   1:  PR[GP1:91,1] = PR[GP1:90,1] + 82.412;
   1:  PR[GP1:91,2] = PR[GP1:90,2] + 125.667;
   1:L PR[91] 10mm/sec FINE;
   1:  PR[GP1:91,1] = PR[GP1:90,1] + 79.591;
   1:  PR[GP1:91,2] = PR[GP1:90,2] + 126.103;
   1:L PR[91] 10mm/sec FINE;
   1:  PR[GP1:91,1] = PR[GP1:90,1] + 77.896;
   1:  PR[GP1:91,2] = PR[GP1:90,2] + 126.057;
   1:L PR[91] 10mm/sec FINE;
   1:  PR[GP1:91,1] = PR[GP1:90,1] + 75.790;
   1:  PR[GP1:91,2] = PR[GP1:90,2] + 125.965;
   1:L PR[91] 10mm/sec FINE;
   1:  PR[GP1:91,1] = PR[GP1:90,1] + 72.240;
   1:  PR[GP1:91,2] = PR[GP1:90,2] + 125.093;
   1:L PR[91] 10mm/sec FINE;
   1:  PR[GP1:91,1] = PR[GP1:90,1] + 68.979;
   1:  PR[GP1:91,2] = PR[GP1:90,2] + 123.554;
   1:L PR[91] 10mm/sec FINE;
   1:  PR[GP1:91,1] = PR[GP1:90,1] + 67.464;
   1:  PR[GP1:91,2] = PR[GP1:90,2] + 122.423;
   1:L PR[91] 10mm/sec FINE;
   1:  PR[GP1:91,1] = PR[GP1:90,1] + 66.133;
   1:  PR[GP1:91,2] = PR[GP1:90,2] + 121.415;
   1:L PR[91] 10mm/sec FINE;
   1:  PR[GP1:91,1] = PR[GP1:90,1] + 63.816;
   1:  PR[GP1:91,2] = PR[GP1:90,2] + 118.763;
   1:L PR[91] 10mm/sec FINE;
   1:  PR[GP1:91,1] = PR[GP1:90,1] + 62.107;
   1:  PR[GP1:91,2] = PR[GP1:90,2] + 115.709;
   1:L PR[91] 10mm/sec FINE;
   1:  PR[GP1:91,1] = PR[GP1:90,1] + 61.054;
   1:  PR[GP1:91,2] = PR[GP1:90,2] + 112.384;
   1:L PR[91] 10mm/sec FINE;
   1:  PR[GP1:91,1] = PR[GP1:90,1] + 60.750;
   1:  PR[GP1:91,2] = PR[GP1:90,2] + 108.893;
   1:L PR[91] 10mm/sec FINE;
   1:  PR[GP1:91,1] = PR[GP1:90,1] + 60.970;
   1:  PR[GP1:91,2] = PR[GP1:90,2] + 107.084;
   1:L PR[91] 10mm/sec FINE;
   1:  PR[GP1:91,1] = PR[GP1:90,1] + 61.204;
   1:  PR[GP1:91,2] = PR[GP1:90,2] + 105.365;
   1:L PR[91] 10mm/sec FINE;
   1:  PR[GP1:91,1] = PR[GP1:90,1] + 62.339;
   1:  PR[GP1:91,2] = PR[GP1:90,2] + 101.980;
   1:L PR[91] 10mm/sec FINE;
   1:  PR[GP1:91,1] = PR[GP1:90,1] + 63.029;
   1:  PR[GP1:91,2] = PR[GP1:90,2] + 100.795;
   1:L PR[91] 10mm/sec FINE;
   1:  PR[GP1:91,1] = PR[GP1:90,1] + 64.194;
   1:  PR[GP1:91,2] = PR[GP1:90,2] + 98.846;
   1:L PR[91] 10mm/sec FINE;
   1:  PR[GP1:91,1] = PR[GP1:90,1] + 64.821;
   1:  PR[GP1:91,2] = PR[GP1:90,2] + 98.140;
   1:L PR[91] 10mm/sec FINE;
   1:  PR[GP1:91,1] = PR[GP1:90,1] + 66.690;
   1:  PR[GP1:91,2] = PR[GP1:90,2] + 96.102;
   1:L PR[91] 10mm/sec FINE;
   1:  PR[GP1:91,1] = PR[GP1:90,1] + 68.560;
   1:  PR[GP1:91,2] = PR[GP1:90,2] + 94.729;
   1:L PR[91] 10mm/sec FINE;
   1:  PR[GP1:91,1] = PR[GP1:90,1] + 69.814;
   1:  PR[GP1:91,2] = PR[GP1:90,2] + 93.845;
   1:L PR[91] 10mm/sec FINE;
   1:  PR[GP1:91,1] = PR[GP1:90,1] + 70.348;
   1:  PR[GP1:91,2] = PR[GP1:90,2] + 93.651;
   1:  PR[GP1:91,3] = PR[GP1:90,3] + 22.900;
   1:L PR[91] 10mm/sec FINE;
   1:  PR[GP1:91,1] = PR[GP1:90,1] + 72.452;
   1:  PR[GP1:91,2] = PR[GP1:90,2] + 92.683;
   1:L PR[91] 10mm/sec FINE;
   1:  PR[GP1:91,1] = PR[GP1:90,1] + 74.148;
   1:  PR[GP1:91,2] = PR[GP1:90,2] + 91.983;
   1:L PR[91] 10mm/sec FINE;
   1:  PR[GP1:91,1] = PR[GP1:90,1] + 75.437;
   1:  PR[GP1:91,2] = PR[GP1:90,2] + 91.661;
   1:L PR[91] 10mm/sec FINE;
   1:  PR[GP1:91,1] = PR[GP1:90,1] + 78.330;
   1:  PR[GP1:91,2] = PR[GP1:90,2] + 91.079;
   1:L PR[91] 10mm/sec FINE;
   1:  PR[GP1:91,1] = PR[GP1:90,1] + 82.087;
   1:  PR[GP1:91,2] = PR[GP1:90,2] + 90.960;
   1:L PR[91] 10mm/sec FINE;
   1:  PR[GP1:91,1] = PR[GP1:90,1] + 83.731;
   1:  PR[GP1:91,2] = PR[GP1:90,2] + 91.115;
   1:L PR[91] 10mm/sec FINE;
   1:  PR[GP1:91,1] = PR[GP1:90,1] + 85.492;
   1:  PR[GP1:91,2] = PR[GP1:90,2] + 91.389;
   1:L PR[91] 10mm/sec FINE;
   1:  PR[GP1:91,1] = PR[GP1:90,1] + 88.274;
   1:  PR[GP1:91,2] = PR[GP1:90,2] + 92.183;
   1:L PR[91] 10mm/sec FINE;
   1:  PR[GP1:91,1] = PR[GP1:90,1] + 88.650;
   1:  PR[GP1:91,2] = PR[GP1:90,2] + 92.270;
   1:L PR[91] 10mm/sec FINE;
   1:  PR[GP1:91,1] = PR[GP1:90,1] + 88.838;
   1:  PR[GP1:91,2] = PR[GP1:90,2] + 92.342;
   1:L PR[91] 10mm/sec FINE;
   1:  PR[GP1:91,1] = PR[GP1:90,1] + 91.683;
   1:  PR[GP1:91,2] = PR[GP1:90,2] + 93.587;
   1:L PR[91] 10mm/sec FINE;
   1:  PR[GP1:91,1] = PR[GP1:90,1] + 93.071;
   1:  PR[GP1:91,2] = PR[GP1:90,2] + 94.392;
   1:L PR[91] 10mm/sec FINE;
   1:  PR[GP1:91,1] = PR[GP1:90,1] + 94.027;
   1:  PR[GP1:91,2] = PR[GP1:90,2] + 95.076;
   1:L PR[91] 10mm/sec FINE;
   1:  PR[GP1:91,1] = PR[GP1:90,1] + 94.243;
   1:  PR[GP1:91,2] = PR[GP1:90,2] + 95.199;
   1:L PR[91] 10mm/sec FINE;
   1:  PR[GP1:91,1] = PR[GP1:90,1] + 94.681;
   1:  PR[GP1:91,2] = PR[GP1:90,2] + 95.389;
   1:L PR[91] 10mm/sec FINE;
   1:  PR[GP1:91,1] = PR[GP1:90,1] + 95.163;
   1:  PR[GP1:91,2] = PR[GP1:90,2] + 95.421;
   1:L PR[91] 10mm/sec FINE;
   1:  PR[GP1:91,1] = PR[GP1:90,1] + 95.410;
   1:  PR[GP1:91,2] = PR[GP1:90,2] + 95.407;
   1:L PR[91] 10mm/sec FINE;
   1:  PR[GP1:91,1] = PR[GP1:90,1] + 95.904;
   1:  PR[GP1:91,2] = PR[GP1:90,2] + 95.271;
   1:L PR[91] 10mm/sec FINE;
   1:  PR[GP1:91,1] = PR[GP1:90,1] + 96.393;
   1:  PR[GP1:91,2] = PR[GP1:90,2] + 94.958;
   1:L PR[91] 10mm/sec FINE;
   1:  PR[GP1:91,1] = PR[GP1:90,1] + 97.232;
   1:  PR[GP1:91,2] = PR[GP1:90,2] + 94.289;
   1:L PR[91] 10mm/sec FINE;
   1:  PR[GP1:91,1] = PR[GP1:90,1] + 97.918;
   1:  PR[GP1:91,2] = PR[GP1:90,2] + 93.780;
   1:L PR[91] 10mm/sec FINE;
   1:  PR[GP1:91,1] = PR[GP1:90,1] + 98.083;
   1:  PR[GP1:91,2] = PR[GP1:90,2] + 93.673;
   1:L PR[91] 10mm/sec FINE;
   1:  PR[GP1:91,1] = PR[GP1:90,1] + 100.385;
   1:  PR[GP1:91,2] = PR[GP1:90,2] + 92.371;
   1:L PR[91] 10mm/sec FINE;
   1:  PR[GP1:91,1] = PR[GP1:90,1] + 102.853;
   1:  PR[GP1:91,2] = PR[GP1:90,2] + 91.430;
   1:L PR[91] 10mm/sec FINE;
   1:  PR[GP1:91,1] = PR[GP1:90,1] + 103.095;
   1:  PR[GP1:91,2] = PR[GP1:90,2] + 91.369;
   1:L PR[91] 10mm/sec FINE;
   1:  PR[GP1:91,1] = PR[GP1:90,1] + 105.479;
   1:  PR[GP1:91,2] = PR[GP1:90,2] + 90.840;
   1:L PR[91] 10mm/sec FINE;
   1:  PR[GP1:91,1] = PR[GP1:90,1] + 106.414;
   1:  PR[GP1:91,2] = PR[GP1:90,2] + 90.749;
   1:L PR[91] 10mm/sec FINE;
   1:  PR[GP1:91,1] = PR[GP1:90,1] + 108.189;
   1:  PR[GP1:91,2] = PR[GP1:90,2] + 90.619;
   1:L PR[91] 10mm/sec FINE;
   1:  PR[GP1:91,1] = PR[GP1:90,1] + 110.016;
   1:  PR[GP1:91,2] = PR[GP1:90,2] + 90.709;
   1:L PR[91] 10mm/sec FINE;
   1:  PR[GP1:91,1] = PR[GP1:90,1] + 110.931;
   1:  PR[GP1:91,2] = PR[GP1:90,2] + 90.772;
   1:L PR[91] 10mm/sec FINE;
   1:  PR[GP1:91,1] = PR[GP1:90,1] + 113.661;
   1:  PR[GP1:91,2] = PR[GP1:90,2] + 91.296;
   1:L PR[91] 10mm/sec FINE;
   1:  PR[GP1:91,1] = PR[GP1:90,1] + 116.348;
   1:  PR[GP1:91,2] = PR[GP1:90,2] + 92.156;
   1:L PR[91] 10mm/sec FINE;
   1:  PR[GP1:91,1] = PR[GP1:90,1] + 117.613;
   1:  PR[GP1:91,2] = PR[GP1:90,2] + 92.742;
   1:L PR[91] 10mm/sec FINE;
   1:  PR[GP1:91,1] = PR[GP1:90,1] + 118.911;
   1:  PR[GP1:91,2] = PR[GP1:90,2] + 93.369;
   1:L PR[91] 10mm/sec FINE;
   1:  PR[GP1:91,1] = PR[GP1:90,1] + 121.140;
   1:  PR[GP1:91,2] = PR[GP1:90,2] + 94.819;
   1:L PR[91] 10mm/sec FINE;
   1:  PR[GP1:91,1] = PR[GP1:90,1] + 121.299;
   1:  PR[GP1:91,2] = PR[GP1:90,2] + 94.926;
   1:L PR[91] 10mm/sec FINE;
   1:  PR[GP1:91,1] = PR[GP1:90,1] + 123.469;
   1:  PR[GP1:91,2] = PR[GP1:90,2] + 96.788;
   1:L PR[91] 10mm/sec FINE;
   1:  PR[GP1:91,1] = PR[GP1:90,1] + 125.338;
   1:  PR[GP1:91,2] = PR[GP1:90,2] + 98.930;
   1:L PR[91] 10mm/sec FINE;
   1:  PR[GP1:91,1] = PR[GP1:90,1] + 126.852;
   1:  PR[GP1:91,2] = PR[GP1:90,2] + 101.311;
   1:L PR[91] 10mm/sec FINE;
   1:  PR[GP1:91,1] = PR[GP1:90,1] + 127.765;
   1:  PR[GP1:91,2] = PR[GP1:90,2] + 103.396;
   1:L PR[91] 10mm/sec FINE;
   1:  PR[GP1:91,1] = PR[GP1:90,1] + 127.971;
   1:  PR[GP1:91,2] = PR[GP1:90,2] + 103.876;
   1:L PR[91] 10mm/sec FINE;
   1:  PR[GP1:91,1] = PR[GP1:90,1] + 128.656;
   1:  PR[GP1:91,2] = PR[GP1:90,2] + 106.564;
   1:L PR[91] 10mm/sec FINE;
   1:  PR[GP1:91,1] = PR[GP1:90,1] + 128.872;
   1:  PR[GP1:91,2] = PR[GP1:90,2] + 109.304;
   1:L PR[91] 10mm/sec FINE;
   1:  PR[GP1:91,1] = PR[GP1:90,1] + 128.474;
   1:  PR[GP1:91,2] = PR[GP1:90,2] + 112.731;
   1:L PR[91] 10mm/sec FINE;
   1:  PR[GP1:91,1] = PR[GP1:90,1] + 127.375;
   1:  PR[GP1:91,2] = PR[GP1:90,2] + 116.010;
   1:L PR[91] 10mm/sec FINE;
   1:  PR[GP1:91,1] = PR[GP1:90,1] + 125.589;
   1:  PR[GP1:91,2] = PR[GP1:90,2] + 119.007;
   1:L PR[91] 10mm/sec FINE;
   1:  PR[GP1:91,1] = PR[GP1:90,1] + 123.186;
   1:  PR[GP1:91,2] = PR[GP1:90,2] + 121.609;
   1:L PR[91] 10mm/sec FINE;
   1:  PR[GP1:91,1] = PR[GP1:90,1] + 120.265;
   1:  PR[GP1:91,2] = PR[GP1:90,2] + 123.714;
   1:L PR[91] 10mm/sec FINE;
   1:  PR[GP1:91,1] = PR[GP1:90,1] + 116.935;
   1:  PR[GP1:91,2] = PR[GP1:90,2] + 125.215;
   1:L PR[91] 10mm/sec FINE;
   1:  PR[GP1:91,1] = PR[GP1:90,1] + 113.317;
   1:  PR[GP1:91,2] = PR[GP1:90,2] + 126.080;
   1:L PR[91] 10mm/sec FINE;
   1:  PR[GP1:91,1] = PR[GP1:90,1] + 112.605;
   1:  PR[GP1:91,2] = PR[GP1:90,2] + 126.119;
   1:L PR[91] 10mm/sec FINE;
   1:  PR[GP1:91,1] = PR[GP1:90,1] + 109.577;
   1:  PR[GP1:91,2] = PR[GP1:90,2] + 126.268;
   1:L PR[91] 10mm/sec FINE;
   1:  PR[GP1:91,1] = PR[GP1:90,1] + 105.878;
   1:  PR[GP1:91,2] = PR[GP1:90,2] + 125.766;
   1:L PR[91] 10mm/sec FINE;
   1:  PR[GP1:91,1] = PR[GP1:90,1] + 102.315;
   1:  PR[GP1:91,2] = PR[GP1:90,2] + 124.617;
   1:L PR[91] 10mm/sec FINE;
   1:  PR[GP1:91,1] = PR[GP1:90,1] + 101.338;
   1:  PR[GP1:91,2] = PR[GP1:90,2] + 124.103;
   1:L PR[91] 10mm/sec FINE;
   1:  PR[GP1:91,1] = PR[GP1:90,1] + 99.069;
   1:  PR[GP1:91,2] = PR[GP1:90,2] + 122.851;
   1:L PR[91] 10mm/sec FINE;
   1:  PR[GP1:91,1] = PR[GP1:90,1] + 96.411;
   1:  PR[GP1:91,2] = PR[GP1:90,2] + 120.730;
   1:L PR[91] 10mm/sec FINE;
   1:  PR[GP1:91,1] = PR[GP1:90,1] + 96.183;
   1:  PR[GP1:91,2] = PR[GP1:90,2] + 120.545;
   1:L PR[91] 10mm/sec FINE;
   1:  PR[GP1:91,1] = PR[GP1:90,1] + 96.101;
   1:  PR[GP1:91,2] = PR[GP1:90,2] + 120.455;
   1:L PR[91] 10mm/sec FINE;
   1:  PR[GP1:91,1] = PR[GP1:90,1] + 95.219;
   1:  PR[GP1:91,2] = PR[GP1:90,2] + 119.857;
   1:L PR[91] 10mm/sec FINE;
   1:  PR[GP1:91,1] = PR[GP1:90,1] + 94.674;
   1:  PR[GP1:91,2] = PR[GP1:90,2] + 119.812;
   1:L PR[91] 10mm/sec FINE;
   1:  PR[GP1:91,1] = PR[GP1:90,1] + 94.127;
   1:  PR[GP1:91,2] = PR[GP1:90,2] + 119.817;
   1:L PR[91] 10mm/sec FINE;
   1:  PR[GP1:91,1] = PR[GP1:90,1] + 93.662;
   1:  PR[GP1:91,2] = PR[GP1:90,2] + 120.062;
   1:L PR[91] 10mm/sec FINE;
   1:  PR[GP1:91,1] = PR[GP1:90,1] + 93.184;
   1:  PR[GP1:91,2] = PR[GP1:90,2] + 120.345;
   1:L PR[91] 10mm/sec FINE;
   1:  PR[GP1:91,1] = PR[GP1:90,1] + 92.028;
   1:  PR[GP1:91,2] = PR[GP1:90,2] + 121.333;
   1:L PR[91] 10mm/sec FINE;
   1:  PR[GP1:91,1] = PR[GP1:90,1] + 90.852;
   1:  PR[GP1:91,2] = PR[GP1:90,2] + 122.143;
   1:L PR[91] 10mm/sec FINE;
   1:  PR[GP1:91,1] = PR[GP1:90,1] + 88.029;
   1:  PR[GP1:91,2] = PR[GP1:90,2] + 123.814;
   1:L PR[91] 10mm/sec FINE;
   1:  PR[GP1:91,1] = PR[GP1:90,1] + 85.285;
   1:  PR[GP1:91,2] = PR[GP1:90,2] + 124.895;
   1:L PR[91] 10mm/sec FINE;
   1:  PR[GP1:91,1] = PR[GP1:90,1] + 84.137;
   1:  PR[GP1:91,2] = PR[GP1:90,2] + 125.299;
   1:L PR[91] 10mm/sec FINE;
   1:  PR[GP1:91,1] = PR[GP1:90,1] + 82.312;
   1:  PR[GP1:91,2] = PR[GP1:90,2] + 125.643;
   1:L PR[91] 10mm/sec FINE;
   1:  PR[GP1:91,1] = PR[GP1:90,1] + 80.128;
   1:  PR[GP1:91,2] = PR[GP1:90,2] + 125.980;
   1:L PR[91] 10mm/sec FINE;
   1:  PR[GP1:91,1] = PR[GP1:90,1] + 79.196;
   1:  PR[GP1:91,2] = PR[GP1:90,2] + 125.975;
   1:L PR[91] 10mm/sec FINE;
   1:  PR[GP1:91,1] = PR[GP1:90,1] + 76.178;
   1:  PR[GP1:91,2] = PR[GP1:90,2] + 125.876;
   1:L PR[91] 10mm/sec FINE;
   1:  PR[GP1:91,1] = PR[GP1:90,1] + 75.062;
   1:  PR[GP1:91,2] = PR[GP1:90,2] + 125.628;
   1:L PR[91] 10mm/sec FINE;
   1:  PR[GP1:91,1] = PR[GP1:90,1] + 72.563;
   1:  PR[GP1:91,2] = PR[GP1:90,2] + 125.016;
   1:L PR[91] 10mm/sec FINE;
   1:  PR[GP1:91,1] = PR[GP1:90,1] + 69.293;
   1:  PR[GP1:91,2] = PR[GP1:90,2] + 123.478;
   1:L PR[91] 10mm/sec FINE;
   1:  PR[GP1:91,1] = PR[GP1:90,1] + 66.439;
   1:  PR[GP1:91,2] = PR[GP1:90,2] + 121.337;
   1:L PR[91] 10mm/sec FINE;
   1:  PR[GP1:91,1] = PR[GP1:90,1] + 64.117;
   1:  PR[GP1:91,2] = PR[GP1:90,2] + 118.682;
   1:L PR[91] 10mm/sec FINE;
   1:  PR[GP1:91,1] = PR[GP1:90,1] + 62.404;
   1:  PR[GP1:91,2] = PR[GP1:90,2] + 115.623;
   1:L PR[91] 10mm/sec FINE;
   1:  PR[GP1:91,1] = PR[GP1:90,1] + 61.348;
   1:  PR[GP1:91,2] = PR[GP1:90,2] + 112.293;
   1:L PR[91] 10mm/sec FINE;
   1:  PR[GP1:91,1] = PR[GP1:90,1] + 61.042;
   1:  PR[GP1:91,2] = PR[GP1:90,2] + 108.795;
   1:L PR[91] 10mm/sec FINE;
   1:  PR[GP1:91,1] = PR[GP1:90,1] + 61.198;
   1:  PR[GP1:91,2] = PR[GP1:90,2] + 107.509;
   1:L PR[91] 10mm/sec FINE;
   1:  PR[GP1:91,1] = PR[GP1:90,1] + 61.227;
   1:  PR[GP1:91,2] = PR[GP1:90,2] + 107.388;
   1:L PR[91] 10mm/sec FINE;
   1:  PR[GP1:91,1] = PR[GP1:90,1] + 61.505;
   1:  PR[GP1:91,2] = PR[GP1:90,2] + 105.256;
   1:L PR[91] 10mm/sec FINE;
   1:  PR[GP1:91,1] = PR[GP1:90,1] + 62.646;
   1:  PR[GP1:91,2] = PR[GP1:90,2] + 101.864;
   1:L PR[91] 10mm/sec FINE;
   1:  PR[GP1:91,1] = PR[GP1:90,1] + 63.080;
   1:  PR[GP1:91,2] = PR[GP1:90,2] + 101.117;
   1:L PR[91] 10mm/sec FINE;
   1:  PR[GP1:91,1] = PR[GP1:90,1] + 64.512;
   1:  PR[GP1:91,2] = PR[GP1:90,2] + 98.723;
   1:L PR[91] 10mm/sec FINE;
   1:  PR[GP1:91,1] = PR[GP1:90,1] + 66.421;
   1:  PR[GP1:91,2] = PR[GP1:90,2] + 96.631;
   1:L PR[91] 10mm/sec FINE;
   1:  PR[GP1:91,1] = PR[GP1:90,1] + 67.065;
   1:  PR[GP1:91,2] = PR[GP1:90,2] + 95.958;
   1:L PR[91] 10mm/sec FINE;
   1:  PR[GP1:91,1] = PR[GP1:90,1] + 69.599;
   1:  PR[GP1:91,2] = PR[GP1:90,2] + 94.149;
   1:L PR[91] 10mm/sec FINE;
   1:  PR[GP1:91,1] = PR[GP1:90,1] + 70.883;
   1:  PR[GP1:91,2] = PR[GP1:90,2] + 93.457;
   1:  PR[GP1:91,3] = PR[GP1:90,3] + 23.900;
   1:L PR[91] 10mm/sec FINE;
   1:  PR[GP1:91,1] = PR[GP1:90,1] + 72.404;
   1:  PR[GP1:91,2] = PR[GP1:90,2] + 92.757;
   1:L PR[91] 10mm/sec FINE;
   1:  PR[GP1:91,1] = PR[GP1:90,1] + 74.729;
   1:  PR[GP1:91,2] = PR[GP1:90,2] + 91.797;
   1:L PR[91] 10mm/sec FINE;
   1:  PR[GP1:91,1] = PR[GP1:90,1] + 75.340;
   1:  PR[GP1:91,2] = PR[GP1:90,2] + 91.644;
   1:L PR[91] 10mm/sec FINE;
   1:  PR[GP1:91,1] = PR[GP1:90,1] + 77.007;
   1:  PR[GP1:91,2] = PR[GP1:90,2] + 91.309;
   1:L PR[91] 10mm/sec FINE;
   1:  PR[GP1:91,1] = PR[GP1:90,1] + 78.702;
   1:  PR[GP1:91,2] = PR[GP1:90,2] + 90.938;
   1:L PR[91] 10mm/sec FINE;
   1:  PR[GP1:91,1] = PR[GP1:90,1] + 79.580;
   1:  PR[GP1:91,2] = PR[GP1:90,2] + 90.864;
   1:L PR[91] 10mm/sec FINE;
   1:  PR[GP1:91,1] = PR[GP1:90,1] + 82.316;
   1:  PR[GP1:91,2] = PR[GP1:90,2] + 90.772;
   1:L PR[91] 10mm/sec FINE;
   1:  PR[GP1:91,1] = PR[GP1:90,1] + 85.126;
   1:  PR[GP1:91,2] = PR[GP1:90,2] + 91.037;
   1:L PR[91] 10mm/sec FINE;
   1:  PR[GP1:91,1] = PR[GP1:90,1] + 85.667;
   1:  PR[GP1:91,2] = PR[GP1:90,2] + 91.121;
   1:L PR[91] 10mm/sec FINE;
   1:  PR[GP1:91,1] = PR[GP1:90,1] + 86.536;
   1:  PR[GP1:91,2] = PR[GP1:90,2] + 91.369;
   1:L PR[91] 10mm/sec FINE;
   1:  PR[GP1:91,1] = PR[GP1:90,1] + 89.160;
   1:  PR[GP1:91,2] = PR[GP1:90,2] + 91.978;
   1:L PR[91] 10mm/sec FINE;
   1:  PR[GP1:91,1] = PR[GP1:90,1] + 90.547;
   1:  PR[GP1:91,2] = PR[GP1:90,2] + 92.510;
   1:L PR[91] 10mm/sec FINE;
   1:  PR[GP1:91,1] = PR[GP1:90,1] + 92.034;
   1:  PR[GP1:91,2] = PR[GP1:90,2] + 93.161;
   1:L PR[91] 10mm/sec FINE;
   1:  PR[GP1:91,1] = PR[GP1:90,1] + 94.287;
   1:  PR[GP1:91,2] = PR[GP1:90,2] + 94.460;
   1:L PR[91] 10mm/sec FINE;
   1:  PR[GP1:91,1] = PR[GP1:90,1] + 94.852;
   1:  PR[GP1:91,2] = PR[GP1:90,2] + 94.701;
   1:L PR[91] 10mm/sec FINE;
   1:  PR[GP1:91,1] = PR[GP1:90,1] + 95.472;
   1:  PR[GP1:91,2] = PR[GP1:90,2] + 94.746;
   1:L PR[91] 10mm/sec FINE;
   1:  PR[GP1:91,1] = PR[GP1:90,1] + 96.183;
   1:  PR[GP1:91,2] = PR[GP1:90,2] + 94.544;
   1:L PR[91] 10mm/sec FINE;
   1:  PR[GP1:91,1] = PR[GP1:90,1] + 96.654;
   1:  PR[GP1:91,2] = PR[GP1:90,2] + 94.264;
   1:L PR[91] 10mm/sec FINE;
   1:  PR[GP1:91,1] = PR[GP1:90,1] + 97.486;
   1:  PR[GP1:91,2] = PR[GP1:90,2] + 93.647;
   1:L PR[91] 10mm/sec FINE;
   1:  PR[GP1:91,1] = PR[GP1:90,1] + 97.858;
   1:  PR[GP1:91,2] = PR[GP1:90,2] + 93.405;
   1:L PR[91] 10mm/sec FINE;
   1:  PR[GP1:91,1] = PR[GP1:90,1] + 99.439;
   1:  PR[GP1:91,2] = PR[GP1:90,2] + 92.506;
   1:L PR[91] 10mm/sec FINE;
   1:  PR[GP1:91,1] = PR[GP1:90,1] + 100.207;
   1:  PR[GP1:91,2] = PR[GP1:90,2] + 92.101;
   1:L PR[91] 10mm/sec FINE;
   1:  PR[GP1:91,1] = PR[GP1:90,1] + 102.242;
   1:  PR[GP1:91,2] = PR[GP1:90,2] + 91.330;
   1:L PR[91] 10mm/sec FINE;
   1:  PR[GP1:91,1] = PR[GP1:90,1] + 102.682;
   1:  PR[GP1:91,2] = PR[GP1:90,2] + 91.182;
   1:L PR[91] 10mm/sec FINE;
   1:  PR[GP1:91,1] = PR[GP1:90,1] + 105.232;
   1:  PR[GP1:91,2] = PR[GP1:90,2] + 90.637;
   1:L PR[91] 10mm/sec FINE;
   1:  PR[GP1:91,1] = PR[GP1:90,1] + 107.945;
   1:  PR[GP1:91,2] = PR[GP1:90,2] + 90.436;
   1:L PR[91] 10mm/sec FINE;
   1:  PR[GP1:91,1] = PR[GP1:90,1] + 108.807;
   1:  PR[GP1:91,2] = PR[GP1:90,2] + 90.479;
   1:L PR[91] 10mm/sec FINE;
   1:  PR[GP1:91,1] = PR[GP1:90,1] + 110.683;
   1:  PR[GP1:91,2] = PR[GP1:90,2] + 90.608;
   1:L PR[91] 10mm/sec FINE;
   1:  PR[GP1:91,1] = PR[GP1:90,1] + 112.522;
   1:  PR[GP1:91,2] = PR[GP1:90,2] + 90.966;
   1:L PR[91] 10mm/sec FINE;
   1:  PR[GP1:91,1] = PR[GP1:90,1] + 113.397;
   1:  PR[GP1:91,2] = PR[GP1:90,2] + 91.152;
   1:L PR[91] 10mm/sec FINE;
   1:  PR[GP1:91,1] = PR[GP1:90,1] + 115.496;
   1:  PR[GP1:91,2] = PR[GP1:90,2] + 91.881;
   1:L PR[91] 10mm/sec FINE;
   1:  PR[GP1:91,1] = PR[GP1:90,1] + 116.048;
   1:  PR[GP1:91,2] = PR[GP1:90,2] + 92.058;
   1:L PR[91] 10mm/sec FINE;
   1:  PR[GP1:91,1] = PR[GP1:90,1] + 118.597;
   1:  PR[GP1:91,2] = PR[GP1:90,2] + 93.285;
   1:L PR[91] 10mm/sec FINE;
   1:  PR[GP1:91,1] = PR[GP1:90,1] + 119.860;
   1:  PR[GP1:91,2] = PR[GP1:90,2] + 94.106;
   1:L PR[91] 10mm/sec FINE;
   1:  PR[GP1:91,1] = PR[GP1:90,1] + 120.965;
   1:  PR[GP1:91,2] = PR[GP1:90,2] + 94.848;
   1:L PR[91] 10mm/sec FINE;
   1:  PR[GP1:91,1] = PR[GP1:90,1] + 123.100;
   1:  PR[GP1:91,2] = PR[GP1:90,2] + 96.728;
   1:L PR[91] 10mm/sec FINE;
   1:  PR[GP1:91,1] = PR[GP1:90,1] + 124.952;
   1:  PR[GP1:91,2] = PR[GP1:90,2] + 98.875;
   1:L PR[91] 10mm/sec FINE;
   1:  PR[GP1:91,1] = PR[GP1:90,1] + 126.455;
   1:  PR[GP1:91,2] = PR[GP1:90,2] + 101.255;
   1:L PR[91] 10mm/sec FINE;
   1:  PR[GP1:91,1] = PR[GP1:90,1] + 127.008;
   1:  PR[GP1:91,2] = PR[GP1:90,2] + 102.520;
   1:L PR[91] 10mm/sec FINE;
   1:  PR[GP1:91,1] = PR[GP1:90,1] + 127.562;
   1:  PR[GP1:91,2] = PR[GP1:90,2] + 103.816;
   1:L PR[91] 10mm/sec FINE;
   1:  PR[GP1:91,1] = PR[GP1:90,1] + 128.240;
   1:  PR[GP1:91,2] = PR[GP1:90,2] + 106.498;
   1:L PR[91] 10mm/sec FINE;
   1:  PR[GP1:91,1] = PR[GP1:90,1] + 128.459;
   1:  PR[GP1:91,2] = PR[GP1:90,2] + 109.240;
   1:L PR[91] 10mm/sec FINE;
   1:  PR[GP1:91,1] = PR[GP1:90,1] + 128.057;
   1:  PR[GP1:91,2] = PR[GP1:90,2] + 112.673;
   1:L PR[91] 10mm/sec FINE;
   1:  PR[GP1:91,1] = PR[GP1:90,1] + 126.952;
   1:  PR[GP1:91,2] = PR[GP1:90,2] + 115.954;
   1:L PR[91] 10mm/sec FINE;
   1:  PR[GP1:91,1] = PR[GP1:90,1] + 125.160;
   1:  PR[GP1:91,2] = PR[GP1:90,2] + 118.952;
   1:L PR[91] 10mm/sec FINE;
   1:  PR[GP1:91,1] = PR[GP1:90,1] + 122.753;
   1:  PR[GP1:91,2] = PR[GP1:90,2] + 121.553;
   1:L PR[91] 10mm/sec FINE;
   1:  PR[GP1:91,1] = PR[GP1:90,1] + 119.826;
   1:  PR[GP1:91,2] = PR[GP1:90,2] + 123.638;
   1:L PR[91] 10mm/sec FINE;
   1:  PR[GP1:91,1] = PR[GP1:90,1] + 116.491;
   1:  PR[GP1:91,2] = PR[GP1:90,2] + 125.132;
   1:L PR[91] 10mm/sec FINE;
   1:  PR[GP1:91,1] = PR[GP1:90,1] + 112.874;
   1:  PR[GP1:91,2] = PR[GP1:90,2] + 125.997;
   1:L PR[91] 10mm/sec FINE;
   1:  PR[GP1:91,1] = PR[GP1:90,1] + 109.156;
   1:  PR[GP1:91,2] = PR[GP1:90,2] + 126.169;
   1:L PR[91] 10mm/sec FINE;
   1:  PR[GP1:91,1] = PR[GP1:90,1] + 105.459;
   1:  PR[GP1:91,2] = PR[GP1:90,2] + 125.665;
   1:L PR[91] 10mm/sec FINE;
   1:  PR[GP1:91,1] = PR[GP1:90,1] + 101.905;
   1:  PR[GP1:91,2] = PR[GP1:90,2] + 124.515;
   1:L PR[91] 10mm/sec FINE;
   1:  PR[GP1:91,1] = PR[GP1:90,1] + 98.679;
   1:  PR[GP1:91,2] = PR[GP1:90,2] + 122.740;
   1:L PR[91] 10mm/sec FINE;
   1:  PR[GP1:91,1] = PR[GP1:90,1] + 96.128;
   1:  PR[GP1:91,2] = PR[GP1:90,2] + 120.716;
   1:L PR[91] 10mm/sec FINE;
   1:  PR[GP1:91,1] = PR[GP1:90,1] + 95.743;
   1:  PR[GP1:91,2] = PR[GP1:90,2] + 120.524;
   1:L PR[91] 10mm/sec FINE;
   1:  PR[GP1:91,1] = PR[GP1:90,1] + 95.243;
   1:  PR[GP1:91,2] = PR[GP1:90,2] + 120.181;
   1:L PR[91] 10mm/sec FINE;
   1:  PR[GP1:91,1] = PR[GP1:90,1] + 94.928;
   1:  PR[GP1:91,2] = PR[GP1:90,2] + 120.155;
   1:L PR[91] 10mm/sec FINE;
   1:  PR[GP1:91,1] = PR[GP1:90,1] + 94.149;
   1:  PR[GP1:91,2] = PR[GP1:90,2] + 120.162;
   1:L PR[91] 10mm/sec FINE;
   1:  PR[GP1:91,1] = PR[GP1:90,1] + 93.313;
   1:  PR[GP1:91,2] = PR[GP1:90,2] + 120.616;
   1:L PR[91] 10mm/sec FINE;
   1:  PR[GP1:91,1] = PR[GP1:90,1] + 92.910;
   1:  PR[GP1:91,2] = PR[GP1:90,2] + 120.959;
   1:L PR[91] 10mm/sec FINE;
   1:  PR[GP1:91,1] = PR[GP1:90,1] + 90.951;
   1:  PR[GP1:91,2] = PR[GP1:90,2] + 122.310;
   1:L PR[91] 10mm/sec FINE;
   1:  PR[GP1:91,1] = PR[GP1:90,1] + 88.917;
   1:  PR[GP1:91,2] = PR[GP1:90,2] + 123.510;
   1:L PR[91] 10mm/sec FINE;
   1:  PR[GP1:91,1] = PR[GP1:90,1] + 88.196;
   1:  PR[GP1:91,2] = PR[GP1:90,2] + 123.838;
   1:L PR[91] 10mm/sec FINE;
   1:  PR[GP1:91,1] = PR[GP1:90,1] + 86.466;
   1:  PR[GP1:91,2] = PR[GP1:90,2] + 124.474;
   1:L PR[91] 10mm/sec FINE;
   1:  PR[GP1:91,1] = PR[GP1:90,1] + 85.189;
   1:  PR[GP1:91,2] = PR[GP1:90,2] + 124.978;
   1:L PR[91] 10mm/sec FINE;
   1:  PR[GP1:91,1] = PR[GP1:90,1] + 84.704;
   1:  PR[GP1:91,2] = PR[GP1:90,2] + 125.148;
   1:L PR[91] 10mm/sec FINE;
   1:  PR[GP1:91,1] = PR[GP1:90,1] + 82.211;
   1:  PR[GP1:91,2] = PR[GP1:90,2] + 125.618;
   1:L PR[91] 10mm/sec FINE;
   1:  PR[GP1:91,1] = PR[GP1:90,1] + 80.668;
   1:  PR[GP1:91,2] = PR[GP1:90,2] + 125.856;
   1:L PR[91] 10mm/sec FINE;
   1:  PR[GP1:91,1] = PR[GP1:90,1] + 79.106;
   1:  PR[GP1:91,2] = PR[GP1:90,2] + 125.849;
   1:L PR[91] 10mm/sec FINE;
   1:  PR[GP1:91,1] = PR[GP1:90,1] + 76.690;
   1:  PR[GP1:91,2] = PR[GP1:90,2] + 125.769;
   1:L PR[91] 10mm/sec FINE;
   1:  PR[GP1:91,1] = PR[GP1:90,1] + 75.946;
   1:  PR[GP1:91,2] = PR[GP1:90,2] + 125.619;
   1:L PR[91] 10mm/sec FINE;
   1:  PR[GP1:91,1] = PR[GP1:90,1] + 72.923;
   1:  PR[GP1:91,2] = PR[GP1:90,2] + 124.933;
   1:L PR[91] 10mm/sec FINE;
   1:  PR[GP1:91,1] = PR[GP1:90,1] + 72.027;
   1:  PR[GP1:91,2] = PR[GP1:90,2] + 124.537;
   1:L PR[91] 10mm/sec FINE;
   1:  PR[GP1:91,1] = PR[GP1:90,1] + 69.607;
   1:  PR[GP1:91,2] = PR[GP1:90,2] + 123.401;
   1:L PR[91] 10mm/sec FINE;
   1:  PR[GP1:91,1] = PR[GP1:90,1] + 66.746;
   1:  PR[GP1:91,2] = PR[GP1:90,2] + 121.259;
   1:L PR[91] 10mm/sec FINE;
   1:  PR[GP1:91,1] = PR[GP1:90,1] + 64.419;
   1:  PR[GP1:91,2] = PR[GP1:90,2] + 118.600;
   1:L PR[91] 10mm/sec FINE;
   1:  PR[GP1:91,1] = PR[GP1:90,1] + 62.702;
   1:  PR[GP1:91,2] = PR[GP1:90,2] + 115.536;
   1:L PR[91] 10mm/sec FINE;
   1:  PR[GP1:91,1] = PR[GP1:90,1] + 61.642;
   1:  PR[GP1:91,2] = PR[GP1:90,2] + 112.201;
   1:L PR[91] 10mm/sec FINE;
   1:  PR[GP1:91,1] = PR[GP1:90,1] + 61.334;
   1:  PR[GP1:91,2] = PR[GP1:90,2] + 108.699;
   1:L PR[91] 10mm/sec FINE;
   1:  PR[GP1:91,1] = PR[GP1:90,1] + 61.806;
   1:  PR[GP1:91,2] = PR[GP1:90,2] + 105.147;
   1:L PR[91] 10mm/sec FINE;
   1:  PR[GP1:91,1] = PR[GP1:90,1] + 62.952;
   1:  PR[GP1:91,2] = PR[GP1:90,2] + 101.747;
   1:L PR[91] 10mm/sec FINE;
   1:  PR[GP1:91,1] = PR[GP1:90,1] + 63.131;
   1:  PR[GP1:91,2] = PR[GP1:90,2] + 101.439;
   1:L PR[91] 10mm/sec FINE;
   1:  PR[GP1:91,1] = PR[GP1:90,1] + 64.475;
   1:  PR[GP1:91,2] = PR[GP1:90,2] + 99.193;
   1:L PR[91] 10mm/sec FINE;
   1:  PR[GP1:91,1] = PR[GP1:90,1] + 64.854;
   1:  PR[GP1:91,2] = PR[GP1:90,2] + 98.592;
   1:L PR[91] 10mm/sec FINE;
   1:  PR[GP1:91,1] = PR[GP1:90,1] + 67.049;
   1:  PR[GP1:91,2] = PR[GP1:90,2] + 96.277;
   1:L PR[91] 10mm/sec FINE;
   1:  PR[GP1:91,1] = PR[GP1:90,1] + 67.561;
   1:  PR[GP1:91,2] = PR[GP1:90,2] + 95.766;
   1:L PR[91] 10mm/sec FINE;
   1:  PR[GP1:91,1] = PR[GP1:90,1] + 69.612;
   1:  PR[GP1:91,2] = PR[GP1:90,2] + 94.302;
   1:L PR[91] 10mm/sec FINE;
   1:  PR[GP1:91,1] = PR[GP1:90,1] + 71.419;
   1:  PR[GP1:91,2] = PR[GP1:90,2] + 93.262;
   1:  PR[GP1:91,3] = PR[GP1:90,3] + 24.900;
   1:L PR[91] 10mm/sec FINE;
   1:  PR[GP1:91,1] = PR[GP1:90,1] + 72.355;
   1:  PR[GP1:91,2] = PR[GP1:90,2] + 92.831;
   1:L PR[91] 10mm/sec FINE;
   1:  PR[GP1:91,1] = PR[GP1:90,1] + 75.295;
   1:  PR[GP1:91,2] = PR[GP1:90,2] + 91.616;
   1:L PR[91] 10mm/sec FINE;
   1:  PR[GP1:91,1] = PR[GP1:90,1] + 75.353;
   1:  PR[GP1:91,2] = PR[GP1:90,2] + 91.601;
   1:L PR[91] 10mm/sec FINE;
   1:  PR[GP1:91,1] = PR[GP1:90,1] + 78.993;
   1:  PR[GP1:91,2] = PR[GP1:90,2] + 90.804;
   1:L PR[91] 10mm/sec FINE;
   1:  PR[GP1:91,1] = PR[GP1:90,1] + 81.018;
   1:  PR[GP1:91,2] = PR[GP1:90,2] + 90.635;
   1:L PR[91] 10mm/sec FINE;
   1:  PR[GP1:91,1] = PR[GP1:90,1] + 82.545;
   1:  PR[GP1:91,2] = PR[GP1:90,2] + 90.584;
   1:L PR[91] 10mm/sec FINE;
   1:  PR[GP1:91,1] = PR[GP1:90,1] + 84.898;
   1:  PR[GP1:91,2] = PR[GP1:90,2] + 90.805;
   1:L PR[91] 10mm/sec FINE;
   1:  PR[GP1:91,1] = PR[GP1:90,1] + 86.147;
   1:  PR[GP1:91,2] = PR[GP1:90,2] + 90.881;
   1:L PR[91] 10mm/sec FINE;
   1:  PR[GP1:91,1] = PR[GP1:90,1] + 89.670;
   1:  PR[GP1:91,2] = PR[GP1:90,2] + 91.687;
   1:L PR[91] 10mm/sec FINE;
   1:  PR[GP1:91,1] = PR[GP1:90,1] + 92.389;
   1:  PR[GP1:91,2] = PR[GP1:90,2] + 92.737;
   1:L PR[91] 10mm/sec FINE;
   1:  PR[GP1:91,1] = PR[GP1:90,1] + 92.584;
   1:  PR[GP1:91,2] = PR[GP1:90,2] + 92.850;
   1:L PR[91] 10mm/sec FINE;
   1:  PR[GP1:91,1] = PR[GP1:90,1] + 94.582;
   1:  PR[GP1:91,2] = PR[GP1:90,2] + 93.882;
   1:L PR[91] 10mm/sec FINE;
   1:  PR[GP1:91,1] = PR[GP1:90,1] + 95.103;
   1:  PR[GP1:91,2] = PR[GP1:90,2] + 94.007;
   1:L PR[91] 10mm/sec FINE;
   1:  PR[GP1:91,1] = PR[GP1:90,1] + 95.334;
   1:  PR[GP1:91,2] = PR[GP1:90,2] + 94.108;
   1:L PR[91] 10mm/sec FINE;
   1:  PR[GP1:91,1] = PR[GP1:90,1] + 95.653;
   1:  PR[GP1:91,2] = PR[GP1:90,2] + 94.131;
   1:L PR[91] 10mm/sec FINE;
   1:  PR[GP1:91,1] = PR[GP1:90,1] + 96.519;
   1:  PR[GP1:91,2] = PR[GP1:90,2] + 93.811;
   1:L PR[91] 10mm/sec FINE;
   1:  PR[GP1:91,1] = PR[GP1:90,1] + 96.691;
   1:  PR[GP1:91,2] = PR[GP1:90,2] + 93.764;
   1:L PR[91] 10mm/sec FINE;
   1:  PR[GP1:91,1] = PR[GP1:90,1] + 97.634;
   1:  PR[GP1:91,2] = PR[GP1:90,2] + 93.137;
   1:L PR[91] 10mm/sec FINE;
   1:  PR[GP1:91,1] = PR[GP1:90,1] + 98.696;
   1:  PR[GP1:91,2] = PR[GP1:90,2] + 92.533;
   1:L PR[91] 10mm/sec FINE;
   1:  PR[GP1:91,1] = PR[GP1:90,1] + 100.032;
   1:  PR[GP1:91,2] = PR[GP1:90,2] + 91.830;
   1:L PR[91] 10mm/sec FINE;
   1:  PR[GP1:91,1] = PR[GP1:90,1] + 101.447;
   1:  PR[GP1:91,2] = PR[GP1:90,2] + 91.294;
   1:L PR[91] 10mm/sec FINE;
   1:  PR[GP1:91,1] = PR[GP1:90,1] + 102.557;
   1:  PR[GP1:91,2] = PR[GP1:90,2] + 90.921;
   1:L PR[91] 10mm/sec FINE;
   1:  PR[GP1:91,1] = PR[GP1:90,1] + 104.463;
   1:  PR[GP1:91,2] = PR[GP1:90,2] + 90.515;
   1:L PR[91] 10mm/sec FINE;
   1:  PR[GP1:91,1] = PR[GP1:90,1] + 105.144;
   1:  PR[GP1:91,2] = PR[GP1:90,2] + 90.402;
   1:L PR[91] 10mm/sec FINE;
   1:  PR[GP1:91,1] = PR[GP1:90,1] + 107.718;
   1:  PR[GP1:91,2] = PR[GP1:90,2] + 90.252;
   1:L PR[91] 10mm/sec FINE;
   1:  PR[GP1:91,1] = PR[GP1:90,1] + 110.435;
   1:  PR[GP1:91,2] = PR[GP1:90,2] + 90.445;
   1:L PR[91] 10mm/sec FINE;
   1:  PR[GP1:91,1] = PR[GP1:90,1] + 111.251;
   1:  PR[GP1:91,2] = PR[GP1:90,2] + 90.604;
   1:L PR[91] 10mm/sec FINE;
   1:  PR[GP1:91,1] = PR[GP1:90,1] + 113.141;
   1:  PR[GP1:91,2] = PR[GP1:90,2] + 91.005;
   1:L PR[91] 10mm/sec FINE;
   1:  PR[GP1:91,1] = PR[GP1:90,1] + 114.982;
   1:  PR[GP1:91,2] = PR[GP1:90,2] + 91.644;
   1:L PR[91] 10mm/sec FINE;
   1:  PR[GP1:91,1] = PR[GP1:90,1] + 115.768;
   1:  PR[GP1:91,2] = PR[GP1:90,2] + 91.931;
   1:L PR[91] 10mm/sec FINE;
   1:  PR[GP1:91,1] = PR[GP1:90,1] + 117.531;
   1:  PR[GP1:91,2] = PR[GP1:90,2] + 92.837;
   1:L PR[91] 10mm/sec FINE;
   1:  PR[GP1:91,1] = PR[GP1:90,1] + 118.280;
   1:  PR[GP1:91,2] = PR[GP1:90,2] + 93.199;
   1:L PR[91] 10mm/sec FINE;
   1:  PR[GP1:91,1] = PR[GP1:90,1] + 120.632;
   1:  PR[GP1:91,2] = PR[GP1:90,2] + 94.771;
   1:L PR[91] 10mm/sec FINE;
   1:  PR[GP1:91,1] = PR[GP1:90,1] + 121.795;
   1:  PR[GP1:91,2] = PR[GP1:90,2] + 95.793;
   1:L PR[91] 10mm/sec FINE;
   1:  PR[GP1:91,1] = PR[GP1:90,1] + 122.747;
   1:  PR[GP1:91,2] = PR[GP1:90,2] + 96.652;
   1:L PR[91] 10mm/sec FINE;
   1:  PR[GP1:91,1] = PR[GP1:90,1] + 124.570;
   1:  PR[GP1:91,2] = PR[GP1:90,2] + 98.814;
   1:L PR[91] 10mm/sec FINE;
   1:  PR[GP1:91,1] = PR[GP1:90,1] + 126.056;
   1:  PR[GP1:91,2] = PR[GP1:90,2] + 101.199;
   1:L PR[91] 10mm/sec FINE;
   1:  PR[GP1:91,1] = PR[GP1:90,1] + 127.154;
   1:  PR[GP1:91,2] = PR[GP1:90,2] + 103.756;
   1:L PR[91] 10mm/sec FINE;
   1:  PR[GP1:91,1] = PR[GP1:90,1] + 127.825;
   1:  PR[GP1:91,2] = PR[GP1:90,2] + 106.431;
   1:L PR[91] 10mm/sec FINE;
   1:  PR[GP1:91,1] = PR[GP1:90,1] + 128.038;
   1:  PR[GP1:91,2] = PR[GP1:90,2] + 109.170;
   1:L PR[91] 10mm/sec FINE;
   1:  PR[GP1:91,1] = PR[GP1:90,1] + 127.639;
   1:  PR[GP1:91,2] = PR[GP1:90,2] + 112.615;
   1:L PR[91] 10mm/sec FINE;
   1:  PR[GP1:91,1] = PR[GP1:90,1] + 126.529;
   1:  PR[GP1:91,2] = PR[GP1:90,2] + 115.897;
   1:L PR[91] 10mm/sec FINE;
   1:  PR[GP1:91,1] = PR[GP1:90,1] + 124.731;
   1:  PR[GP1:91,2] = PR[GP1:90,2] + 118.897;
   1:L PR[91] 10mm/sec FINE;
   1:  PR[GP1:91,1] = PR[GP1:90,1] + 124.127;
   1:  PR[GP1:91,2] = PR[GP1:90,2] + 119.548;
   1:L PR[91] 10mm/sec FINE;
   1:  PR[GP1:91,1] = PR[GP1:90,1] + 122.318;
   1:  PR[GP1:91,2] = PR[GP1:90,2] + 121.479;
   1:L PR[91] 10mm/sec FINE;
   1:  PR[GP1:91,1] = PR[GP1:90,1] + 119.387;
   1:  PR[GP1:91,2] = PR[GP1:90,2] + 123.552;
   1:L PR[91] 10mm/sec FINE;
   1:  PR[GP1:91,1] = PR[GP1:90,1] + 116.047;
   1:  PR[GP1:91,2] = PR[GP1:90,2] + 125.049;
   1:L PR[91] 10mm/sec FINE;
   1:  PR[GP1:91,1] = PR[GP1:90,1] + 112.460;
   1:  PR[GP1:91,2] = PR[GP1:90,2] + 125.891;
   1:L PR[91] 10mm/sec FINE;
   1:  PR[GP1:91,1] = PR[GP1:90,1] + 110.047;
   1:  PR[GP1:91,2] = PR[GP1:90,2] + 126.005;
   1:L PR[91] 10mm/sec FINE;
   1:  PR[GP1:91,1] = PR[GP1:90,1] + 108.755;
   1:  PR[GP1:91,2] = PR[GP1:90,2] + 126.059;
   1:L PR[91] 10mm/sec FINE;
   1:  PR[GP1:91,1] = PR[GP1:90,1] + 105.041;
   1:  PR[GP1:91,2] = PR[GP1:90,2] + 125.564;
   1:L PR[91] 10mm/sec FINE;
   1:  PR[GP1:91,1] = PR[GP1:90,1] + 101.546;
   1:  PR[GP1:91,2] = PR[GP1:90,2] + 124.394;
   1:L PR[91] 10mm/sec FINE;
   1:  PR[GP1:91,1] = PR[GP1:90,1] + 98.289;
   1:  PR[GP1:91,2] = PR[GP1:90,2] + 122.629;
   1:L PR[91] 10mm/sec FINE;
   1:  PR[GP1:91,1] = PR[GP1:90,1] + 96.188;
   1:  PR[GP1:91,2] = PR[GP1:90,2] + 120.979;
   1:L PR[91] 10mm/sec FINE;
   1:  PR[GP1:91,1] = PR[GP1:90,1] + 95.244;
   1:  PR[GP1:91,2] = PR[GP1:90,2] + 120.500;
   1:L PR[91] 10mm/sec FINE;
   1:  PR[GP1:91,1] = PR[GP1:90,1] + 94.177;
   1:  PR[GP1:91,2] = PR[GP1:90,2] + 120.508;
   1:L PR[91] 10mm/sec FINE;
   1:  PR[GP1:91,1] = PR[GP1:90,1] + 93.473;
   1:  PR[GP1:91,2] = PR[GP1:90,2] + 120.855;
   1:L PR[91] 10mm/sec FINE;
   1:  PR[GP1:91,1] = PR[GP1:90,1] + 92.859;
   1:  PR[GP1:91,2] = PR[GP1:90,2] + 121.229;
   1:L PR[91] 10mm/sec FINE;
   1:  PR[GP1:91,1] = PR[GP1:90,1] + 91.050;
   1:  PR[GP1:91,2] = PR[GP1:90,2] + 122.476;
   1:L PR[91] 10mm/sec FINE;
   1:  PR[GP1:91,1] = PR[GP1:90,1] + 89.837;
   1:  PR[GP1:91,2] = PR[GP1:90,2] + 123.192;
   1:L PR[91] 10mm/sec FINE;
   1:  PR[GP1:91,1] = PR[GP1:90,1] + 88.311;
   1:  PR[GP1:91,2] = PR[GP1:90,2] + 123.887;
   1:L PR[91] 10mm/sec FINE;
   1:  PR[GP1:91,1] = PR[GP1:90,1] + 85.363;
   1:  PR[GP1:91,2] = PR[GP1:90,2] + 124.971;
   1:L PR[91] 10mm/sec FINE;
   1:  PR[GP1:91,1] = PR[GP1:90,1] + 85.178;
   1:  PR[GP1:91,2] = PR[GP1:90,2] + 125.021;
   1:L PR[91] 10mm/sec FINE;
   1:  PR[GP1:91,1] = PR[GP1:90,1] + 82.110;
   1:  PR[GP1:91,2] = PR[GP1:90,2] + 125.593;
   1:L PR[91] 10mm/sec FINE;
   1:  PR[GP1:91,1] = PR[GP1:90,1] + 81.208;
   1:  PR[GP1:91,2] = PR[GP1:90,2] + 125.732;
   1:L PR[91] 10mm/sec FINE;
   1:  PR[GP1:91,1] = PR[GP1:90,1] + 79.017;
   1:  PR[GP1:91,2] = PR[GP1:90,2] + 125.722;
   1:L PR[91] 10mm/sec FINE;
   1:  PR[GP1:91,1] = PR[GP1:90,1] + 77.203;
   1:  PR[GP1:91,2] = PR[GP1:90,2] + 125.662;
   1:L PR[91] 10mm/sec FINE;
   1:  PR[GP1:91,1] = PR[GP1:90,1] + 75.882;
   1:  PR[GP1:91,2] = PR[GP1:90,2] + 125.395;
   1:L PR[91] 10mm/sec FINE;
   1:  PR[GP1:91,1] = PR[GP1:90,1] + 73.411;
   1:  PR[GP1:91,2] = PR[GP1:90,2] + 124.835;
   1:L PR[91] 10mm/sec FINE;
   1:  PR[GP1:91,1] = PR[GP1:90,1] + 72.790;
   1:  PR[GP1:91,2] = PR[GP1:90,2] + 124.573;
   1:L PR[91] 10mm/sec FINE;
   1:  PR[GP1:91,1] = PR[GP1:90,1] + 69.967;
   1:  PR[GP1:91,2] = PR[GP1:90,2] + 123.317;
   1:L PR[91] 10mm/sec FINE;
   1:  PR[GP1:91,1] = PR[GP1:90,1] + 68.674;
   1:  PR[GP1:91,2] = PR[GP1:90,2] + 122.393;
   1:L PR[91] 10mm/sec FINE;
   1:  PR[GP1:91,1] = PR[GP1:90,1] + 67.053;
   1:  PR[GP1:91,2] = PR[GP1:90,2] + 121.181;
   1:L PR[91] 10mm/sec FINE;
   1:  PR[GP1:91,1] = PR[GP1:90,1] + 64.720;
   1:  PR[GP1:91,2] = PR[GP1:90,2] + 118.519;
   1:L PR[91] 10mm/sec FINE;
   1:  PR[GP1:91,1] = PR[GP1:90,1] + 62.999;
   1:  PR[GP1:91,2] = PR[GP1:90,2] + 115.450;
   1:L PR[91] 10mm/sec FINE;
   1:  PR[GP1:91,1] = PR[GP1:90,1] + 61.935;
   1:  PR[GP1:91,2] = PR[GP1:90,2] + 112.110;
   1:L PR[91] 10mm/sec FINE;
   1:  PR[GP1:91,1] = PR[GP1:90,1] + 61.626;
   1:  PR[GP1:91,2] = PR[GP1:90,2] + 108.601;
   1:L PR[91] 10mm/sec FINE;
   1:  PR[GP1:91,1] = PR[GP1:90,1] + 61.658;
   1:  PR[GP1:91,2] = PR[GP1:90,2] + 108.339;
   1:L PR[91] 10mm/sec FINE;
   1:  PR[GP1:91,1] = PR[GP1:90,1] + 61.699;
   1:  PR[GP1:91,2] = PR[GP1:90,2] + 108.162;
   1:L PR[91] 10mm/sec FINE;
   1:  PR[GP1:91,1] = PR[GP1:90,1] + 62.107;
   1:  PR[GP1:91,2] = PR[GP1:90,2] + 105.038;
   1:L PR[91] 10mm/sec FINE;
   1:  PR[GP1:91,1] = PR[GP1:90,1] + 62.849;
   1:  PR[GP1:91,2] = PR[GP1:90,2] + 102.841;
   1:L PR[91] 10mm/sec FINE;
   1:  PR[GP1:91,1] = PR[GP1:90,1] + 63.251;
   1:  PR[GP1:91,2] = PR[GP1:90,2] + 101.729;
   1:L PR[91] 10mm/sec FINE;
   1:  PR[GP1:91,1] = PR[GP1:90,1] + 63.291;
   1:  PR[GP1:91,2] = PR[GP1:90,2] + 101.623;
   1:L PR[91] 10mm/sec FINE;
   1:  PR[GP1:91,1] = PR[GP1:90,1] + 64.972;
   1:  PR[GP1:91,2] = PR[GP1:90,2] + 98.939;
   1:L PR[91] 10mm/sec FINE;
   1:  PR[GP1:91,1] = PR[GP1:90,1] + 65.320;
   1:  PR[GP1:91,2] = PR[GP1:90,2] + 98.408;
   1:L PR[91] 10mm/sec FINE;
   1:  PR[GP1:91,1] = PR[GP1:90,1] + 67.131;
   1:  PR[GP1:91,2] = PR[GP1:90,2] + 96.499;
   1:L PR[91] 10mm/sec FINE;
   1:  PR[GP1:91,1] = PR[GP1:90,1] + 68.060;
   1:  PR[GP1:91,2] = PR[GP1:90,2] + 95.572;
   1:L PR[91] 10mm/sec FINE;
   1:  PR[GP1:91,1] = PR[GP1:90,1] + 69.624;
   1:  PR[GP1:91,2] = PR[GP1:90,2] + 94.455;
   1:L PR[91] 10mm/sec FINE;
   1:  PR[GP1:91,1] = PR[GP1:90,1] + 71.955;
   1:  PR[GP1:91,2] = PR[GP1:90,2] + 93.067;
   1:  PR[GP1:91,3] = PR[GP1:90,3] + 25.900;
   1:L PR[91] 10mm/sec FINE;
   1:  PR[GP1:91,1] = PR[GP1:90,1] + 72.308;
   1:  PR[GP1:91,2] = PR[GP1:90,2] + 92.904;
   1:L PR[91] 10mm/sec FINE;
   1:  PR[GP1:91,1] = PR[GP1:90,1] + 75.650;
   1:  PR[GP1:91,2] = PR[GP1:90,2] + 91.515;
   1:L PR[91] 10mm/sec FINE;
   1:  PR[GP1:91,1] = PR[GP1:90,1] + 76.779;
   1:  PR[GP1:91,2] = PR[GP1:90,2] + 91.219;
   1:L PR[91] 10mm/sec FINE;
   1:  PR[GP1:91,1] = PR[GP1:90,1] + 79.284;
   1:  PR[GP1:91,2] = PR[GP1:90,2] + 90.671;
   1:L PR[91] 10mm/sec FINE;
   1:  PR[GP1:91,1] = PR[GP1:90,1] + 82.455;
   1:  PR[GP1:91,2] = PR[GP1:90,2] + 90.407;
   1:L PR[91] 10mm/sec FINE;
   1:  PR[GP1:91,1] = PR[GP1:90,1] + 82.774;
   1:  PR[GP1:91,2] = PR[GP1:90,2] + 90.396;
   1:L PR[91] 10mm/sec FINE;
   1:  PR[GP1:91,1] = PR[GP1:90,1] + 83.281;
   1:  PR[GP1:91,2] = PR[GP1:90,2] + 90.443;
   1:L PR[91] 10mm/sec FINE;
   1:  PR[GP1:91,1] = PR[GP1:90,1] + 85.888;
   1:  PR[GP1:91,2] = PR[GP1:90,2] + 90.592;
   1:L PR[91] 10mm/sec FINE;
   1:  PR[GP1:91,1] = PR[GP1:90,1] + 86.858;
   1:  PR[GP1:91,2] = PR[GP1:90,2] + 90.661;
   1:L PR[91] 10mm/sec FINE;
   1:  PR[GP1:91,1] = PR[GP1:90,1] + 90.180;
   1:  PR[GP1:91,2] = PR[GP1:90,2] + 91.395;
   1:L PR[91] 10mm/sec FINE;
   1:  PR[GP1:91,1] = PR[GP1:90,1] + 91.149;
   1:  PR[GP1:91,2] = PR[GP1:90,2] + 91.767;
   1:L PR[91] 10mm/sec FINE;
   1:  PR[GP1:91,1] = PR[GP1:90,1] + 93.091;
   1:  PR[GP1:91,2] = PR[GP1:90,2] + 92.423;
   1:L PR[91] 10mm/sec FINE;
   1:  PR[GP1:91,1] = PR[GP1:90,1] + 93.553;
   1:  PR[GP1:91,2] = PR[GP1:90,2] + 92.641;
   1:L PR[91] 10mm/sec FINE;
   1:  PR[GP1:91,1] = PR[GP1:90,1] + 94.864;
   1:  PR[GP1:91,2] = PR[GP1:90,2] + 93.304;
   1:L PR[91] 10mm/sec FINE;
   1:  PR[GP1:91,1] = PR[GP1:90,1] + 95.811;
   1:  PR[GP1:91,2] = PR[GP1:90,2] + 93.532;
   1:L PR[91] 10mm/sec FINE;
   1:  PR[GP1:91,1] = PR[GP1:90,1] + 97.001;
   1:  PR[GP1:91,2] = PR[GP1:90,2] + 93.135;
   1:L PR[91] 10mm/sec FINE;
   1:  PR[GP1:91,1] = PR[GP1:90,1] + 97.409;
   1:  PR[GP1:91,2] = PR[GP1:90,2] + 92.870;
   1:L PR[91] 10mm/sec FINE;
   1:  PR[GP1:91,1] = PR[GP1:90,1] + 97.939;
   1:  PR[GP1:91,2] = PR[GP1:90,2] + 92.568;
   1:L PR[91] 10mm/sec FINE;
   1:  PR[GP1:91,1] = PR[GP1:90,1] + 99.856;
   1:  PR[GP1:91,2] = PR[GP1:90,2] + 91.558;
   1:L PR[91] 10mm/sec FINE;
   1:  PR[GP1:91,1] = PR[GP1:90,1] + 100.652;
   1:  PR[GP1:91,2] = PR[GP1:90,2] + 91.257;
   1:L PR[91] 10mm/sec FINE;
   1:  PR[GP1:91,1] = PR[GP1:90,1] + 102.433;
   1:  PR[GP1:91,2] = PR[GP1:90,2] + 90.659;
   1:L PR[91] 10mm/sec FINE;
   1:  PR[GP1:91,1] = PR[GP1:90,1] + 103.645;
   1:  PR[GP1:91,2] = PR[GP1:90,2] + 90.402;
   1:L PR[91] 10mm/sec FINE;
   1:  PR[GP1:91,1] = PR[GP1:90,1] + 105.074;
   1:  PR[GP1:91,2] = PR[GP1:90,2] + 90.163;
   1:L PR[91] 10mm/sec FINE;
   1:  PR[GP1:91,1] = PR[GP1:90,1] + 106.826;
   1:  PR[GP1:91,2] = PR[GP1:90,2] + 90.059;
   1:L PR[91] 10mm/sec FINE;
   1:  PR[GP1:91,1] = PR[GP1:90,1] + 107.695;
   1:  PR[GP1:91,2] = PR[GP1:90,2] + 90.050;
   1:L PR[91] 10mm/sec FINE;
   1:  PR[GP1:91,1] = PR[GP1:90,1] + 110.236;
   1:  PR[GP1:91,2] = PR[GP1:90,2] + 90.283;
   1:L PR[91] 10mm/sec FINE;
   1:  PR[GP1:91,1] = PR[GP1:90,1] + 112.884;
   1:  PR[GP1:91,2] = PR[GP1:90,2] + 90.858;
   1:L PR[91] 10mm/sec FINE;
   1:  PR[GP1:91,1] = PR[GP1:90,1] + 115.501;
   1:  PR[GP1:91,2] = PR[GP1:90,2] + 91.797;
   1:L PR[91] 10mm/sec FINE;
   1:  PR[GP1:91,1] = PR[GP1:90,1] + 117.984;
   1:  PR[GP1:91,2] = PR[GP1:90,2] + 93.085;
   1:L PR[91] 10mm/sec FINE;
   1:  PR[GP1:91,1] = PR[GP1:90,1] + 119.459;
   1:  PR[GP1:91,2] = PR[GP1:90,2] + 94.130;
   1:L PR[91] 10mm/sec FINE;
   1:  PR[GP1:91,1] = PR[GP1:90,1] + 120.298;
   1:  PR[GP1:91,2] = PR[GP1:90,2] + 94.693;
   1:L PR[91] 10mm/sec FINE;
   1:  PR[GP1:91,1] = PR[GP1:90,1] + 122.395;
   1:  PR[GP1:91,2] = PR[GP1:90,2] + 96.577;
   1:L PR[91] 10mm/sec FINE;
   1:  PR[GP1:91,1] = PR[GP1:90,1] + 124.200;
   1:  PR[GP1:91,2] = PR[GP1:90,2] + 98.737;
   1:L PR[91] 10mm/sec FINE;
   1:  PR[GP1:91,1] = PR[GP1:90,1] + 125.437;
   1:  PR[GP1:91,2] = PR[GP1:90,2] + 100.752;
   1:L PR[91] 10mm/sec FINE;
   1:  PR[GP1:91,1] = PR[GP1:90,1] + 125.663;
   1:  PR[GP1:91,2] = PR[GP1:90,2] + 101.129;
   1:L PR[91] 10mm/sec FINE;
   1:  PR[GP1:91,1] = PR[GP1:90,1] + 126.746;
   1:  PR[GP1:91,2] = PR[GP1:90,2] + 103.695;
   1:L PR[91] 10mm/sec FINE;
   1:  PR[GP1:91,1] = PR[GP1:90,1] + 127.409;
   1:  PR[GP1:91,2] = PR[GP1:90,2] + 106.365;
   1:L PR[91] 10mm/sec FINE;
   1:  PR[GP1:91,1] = PR[GP1:90,1] + 127.617;
   1:  PR[GP1:91,2] = PR[GP1:90,2] + 109.100;
   1:L PR[91] 10mm/sec FINE;
   1:  PR[GP1:91,1] = PR[GP1:90,1] + 127.220;
   1:  PR[GP1:91,2] = PR[GP1:90,2] + 112.549;
   1:L PR[91] 10mm/sec FINE;
   1:  PR[GP1:91,1] = PR[GP1:90,1] + 126.104;
   1:  PR[GP1:91,2] = PR[GP1:90,2] + 115.829;
   1:L PR[91] 10mm/sec FINE;
   1:  PR[GP1:91,1] = PR[GP1:90,1] + 124.301;
   1:  PR[GP1:91,2] = PR[GP1:90,2] + 118.814;
   1:L PR[91] 10mm/sec FINE;
   1:  PR[GP1:91,1] = PR[GP1:90,1] + 121.883;
   1:  PR[GP1:91,2] = PR[GP1:90,2] + 121.392;
   1:L PR[91] 10mm/sec FINE;
   1:  PR[GP1:91,1] = PR[GP1:90,1] + 118.947;
   1:  PR[GP1:91,2] = PR[GP1:90,2] + 123.467;
   1:L PR[91] 10mm/sec FINE;
   1:  PR[GP1:91,1] = PR[GP1:90,1] + 115.613;
   1:  PR[GP1:91,2] = PR[GP1:90,2] + 124.959;
   1:L PR[91] 10mm/sec FINE;
   1:  PR[GP1:91,1] = PR[GP1:90,1] + 112.047;
   1:  PR[GP1:91,2] = PR[GP1:90,2] + 125.785;
   1:L PR[91] 10mm/sec FINE;
   1:  PR[GP1:91,1] = PR[GP1:90,1] + 108.353;
   1:  PR[GP1:91,2] = PR[GP1:90,2] + 125.948;
   1:L PR[91] 10mm/sec FINE;
   1:  PR[GP1:91,1] = PR[GP1:90,1] + 105.914;
   1:  PR[GP1:91,2] = PR[GP1:90,2] + 125.624;
   1:L PR[91] 10mm/sec FINE;
   1:  PR[GP1:91,1] = PR[GP1:90,1] + 104.679;
   1:  PR[GP1:91,2] = PR[GP1:90,2] + 125.441;
   1:L PR[91] 10mm/sec FINE;
   1:  PR[GP1:91,1] = PR[GP1:90,1] + 101.186;
   1:  PR[GP1:91,2] = PR[GP1:90,2] + 124.272;
   1:L PR[91] 10mm/sec FINE;
   1:  PR[GP1:91,1] = PR[GP1:90,1] + 98.641;
   1:  PR[GP1:91,2] = PR[GP1:90,2] + 122.899;
   1:L PR[91] 10mm/sec FINE;
   1:  PR[GP1:91,1] = PR[GP1:90,1] + 97.954;
   1:  PR[GP1:91,2] = PR[GP1:90,2] + 122.507;
   1:L PR[91] 10mm/sec FINE;
   1:  PR[GP1:91,1] = PR[GP1:90,1] + 96.251;
   1:  PR[GP1:91,2] = PR[GP1:90,2] + 121.236;
   1:L PR[91] 10mm/sec FINE;
   1:  PR[GP1:91,1] = PR[GP1:90,1] + 95.291;
   1:  PR[GP1:91,2] = PR[GP1:90,2] + 120.724;
   1:L PR[91] 10mm/sec FINE;
   1:  PR[GP1:91,1] = PR[GP1:90,1] + 95.072;
   1:  PR[GP1:91,2] = PR[GP1:90,2] + 120.754;
   1:L PR[91] 10mm/sec FINE;
   1:  PR[GP1:91,1] = PR[GP1:90,1] + 94.255;
   1:  PR[GP1:91,2] = PR[GP1:90,2] + 120.769;
   1:L PR[91] 10mm/sec FINE;
   1:  PR[GP1:91,1] = PR[GP1:90,1] + 93.629;
   1:  PR[GP1:91,2] = PR[GP1:90,2] + 121.086;
   1:L PR[91] 10mm/sec FINE;
   1:  PR[GP1:91,1] = PR[GP1:90,1] + 91.749;
   1:  PR[GP1:91,2] = PR[GP1:90,2] + 122.229;
   1:L PR[91] 10mm/sec FINE;
   1:  PR[GP1:91,1] = PR[GP1:90,1] + 91.150;
   1:  PR[GP1:91,2] = PR[GP1:90,2] + 122.642;
   1:L PR[91] 10mm/sec FINE;
   1:  PR[GP1:91,1] = PR[GP1:90,1] + 90.757;
   1:  PR[GP1:91,2] = PR[GP1:90,2] + 122.874;
   1:L PR[91] 10mm/sec FINE;
   1:  PR[GP1:91,1] = PR[GP1:90,1] + 88.426;
   1:  PR[GP1:91,2] = PR[GP1:90,2] + 123.936;
   1:L PR[91] 10mm/sec FINE;
   1:  PR[GP1:91,1] = PR[GP1:90,1] + 86.350;
   1:  PR[GP1:91,2] = PR[GP1:90,2] + 124.700;
   1:L PR[91] 10mm/sec FINE;
   1:  PR[GP1:91,1] = PR[GP1:90,1] + 85.330;
   1:  PR[GP1:91,2] = PR[GP1:90,2] + 124.972;
   1:L PR[91] 10mm/sec FINE;
   1:  PR[GP1:91,1] = PR[GP1:90,1] + 81.746;
   1:  PR[GP1:91,2] = PR[GP1:90,2] + 125.609;
   1:L PR[91] 10mm/sec FINE;
   1:  PR[GP1:91,1] = PR[GP1:90,1] + 78.928;
   1:  PR[GP1:91,2] = PR[GP1:90,2] + 125.595;
   1:L PR[91] 10mm/sec FINE;
   1:  PR[GP1:91,1] = PR[GP1:90,1] + 77.716;
   1:  PR[GP1:91,2] = PR[GP1:90,2] + 125.556;
   1:L PR[91] 10mm/sec FINE;
   1:  PR[GP1:91,1] = PR[GP1:90,1] + 75.819;
   1:  PR[GP1:91,2] = PR[GP1:90,2] + 125.172;
   1:L PR[91] 10mm/sec FINE;
   1:  PR[GP1:91,1] = PR[GP1:90,1] + 73.900;
   1:  PR[GP1:91,2] = PR[GP1:90,2] + 124.737;
   1:L PR[91] 10mm/sec FINE;
   1:  PR[GP1:91,1] = PR[GP1:90,1] + 72.765;
   1:  PR[GP1:91,2] = PR[GP1:90,2] + 124.258;
   1:L PR[91] 10mm/sec FINE;
   1:  PR[GP1:91,1] = PR[GP1:90,1] + 70.433;
   1:  PR[GP1:91,2] = PR[GP1:90,2] + 123.220;
   1:L PR[91] 10mm/sec FINE;
   1:  PR[GP1:91,1] = PR[GP1:90,1] + 69.869;
   1:  PR[GP1:91,2] = PR[GP1:90,2] + 122.828;
   1:L PR[91] 10mm/sec FINE;
   1:  PR[GP1:91,1] = PR[GP1:90,1] + 67.440;
   1:  PR[GP1:91,2] = PR[GP1:90,2] + 121.089;
   1:L PR[91] 10mm/sec FINE;
   1:  PR[GP1:91,1] = PR[GP1:90,1] + 65.031;
   1:  PR[GP1:91,2] = PR[GP1:90,2] + 118.433;
   1:L PR[91] 10mm/sec FINE;
   1:  PR[GP1:91,1] = PR[GP1:90,1] + 63.297;
   1:  PR[GP1:91,2] = PR[GP1:90,2] + 115.363;
   1:L PR[91] 10mm/sec FINE;
   1:  PR[GP1:91,1] = PR[GP1:90,1] + 62.229;
   1:  PR[GP1:91,2] = PR[GP1:90,2] + 112.018;
   1:L PR[91] 10mm/sec FINE;
   1:  PR[GP1:91,1] = PR[GP1:90,1] + 62.127;
   1:  PR[GP1:91,2] = PR[GP1:90,2] + 110.860;
   1:L PR[91] 10mm/sec FINE;
   1:  PR[GP1:91,1] = PR[GP1:90,1] + 61.990;
   1:  PR[GP1:91,2] = PR[GP1:90,2] + 109.080;
   1:L PR[91] 10mm/sec FINE;
   1:  PR[GP1:91,1] = PR[GP1:90,1] + 61.948;
   1:  PR[GP1:91,2] = PR[GP1:90,2] + 108.498;
   1:L PR[91] 10mm/sec FINE;
   1:  PR[GP1:91,1] = PR[GP1:90,1] + 62.479;
   1:  PR[GP1:91,2] = PR[GP1:90,2] + 104.907;
   1:L PR[91] 10mm/sec FINE;
   1:  PR[GP1:91,1] = PR[GP1:90,1] + 63.737;
   1:  PR[GP1:91,2] = PR[GP1:90,2] + 101.450;
   1:L PR[91] 10mm/sec FINE;
   1:  PR[GP1:91,1] = PR[GP1:90,1] + 65.134;
   1:  PR[GP1:91,2] = PR[GP1:90,2] + 99.219;
   1:L PR[91] 10mm/sec FINE;
   1:  PR[GP1:91,1] = PR[GP1:90,1] + 65.788;
   1:  PR[GP1:91,2] = PR[GP1:90,2] + 98.223;
   1:L PR[91] 10mm/sec FINE;
   1:  PR[GP1:91,1] = PR[GP1:90,1] + 67.213;
   1:  PR[GP1:91,2] = PR[GP1:90,2] + 96.721;
   1:L PR[91] 10mm/sec FINE;
   1:  PR[GP1:91,1] = PR[GP1:90,1] + 68.558;
   1:  PR[GP1:91,2] = PR[GP1:90,2] + 95.378;
   1:L PR[91] 10mm/sec FINE;
   1:  PR[GP1:91,1] = PR[GP1:90,1] + 69.636;
   1:  PR[GP1:91,2] = PR[GP1:90,2] + 94.608;
   1:L PR[91] 10mm/sec FINE;
   1:  PR[GP1:91,1] = PR[GP1:90,1] + 72.446;
   1:  PR[GP1:91,2] = PR[GP1:90,2] + 92.911;
   1:  PR[GP1:91,3] = PR[GP1:90,3] + 26.900;
   1:L PR[91] 10mm/sec FINE;
   1:  PR[GP1:91,1] = PR[GP1:90,1] + 72.776;
   1:  PR[GP1:91,2] = PR[GP1:90,2] + 92.760;
   1:L PR[91] 10mm/sec FINE;
   1:  PR[GP1:91,1] = PR[GP1:90,1] + 76.005;
   1:  PR[GP1:91,2] = PR[GP1:90,2] + 91.414;
   1:L PR[91] 10mm/sec FINE;
   1:  PR[GP1:91,1] = PR[GP1:90,1] + 78.206;
   1:  PR[GP1:91,2] = PR[GP1:90,2] + 90.837;
   1:L PR[91] 10mm/sec FINE;
   1:  PR[GP1:91,1] = PR[GP1:90,1] + 79.576;
   1:  PR[GP1:91,2] = PR[GP1:90,2] + 90.537;
   1:L PR[91] 10mm/sec FINE;
   1:  PR[GP1:91,1] = PR[GP1:90,1] + 81.771;
   1:  PR[GP1:91,2] = PR[GP1:90,2] + 90.354;
   1:L PR[91] 10mm/sec FINE;
   1:  PR[GP1:91,1] = PR[GP1:90,1] + 83.016;
   1:  PR[GP1:91,2] = PR[GP1:90,2] + 90.216;
   1:L PR[91] 10mm/sec FINE;
   1:  PR[GP1:91,1] = PR[GP1:90,1] + 83.530;
   1:  PR[GP1:91,2] = PR[GP1:90,2] + 90.188;
   1:L PR[91] 10mm/sec FINE;
   1:  PR[GP1:91,1] = PR[GP1:90,1] + 85.960;
   1:  PR[GP1:91,2] = PR[GP1:90,2] + 90.326;
   1:L PR[91] 10mm/sec FINE;
   1:  PR[GP1:91,1] = PR[GP1:90,1] + 87.570;
   1:  PR[GP1:91,2] = PR[GP1:90,2] + 90.441;
   1:L PR[91] 10mm/sec FINE;
   1:  PR[GP1:91,1] = PR[GP1:90,1] + 89.775;
   1:  PR[GP1:91,2] = PR[GP1:90,2] + 90.919;
   1:L PR[91] 10mm/sec FINE;
   1:  PR[GP1:91,1] = PR[GP1:90,1] + 90.871;
   1:  PR[GP1:91,2] = PR[GP1:90,2] + 91.114;
   1:L PR[91] 10mm/sec FINE;
   1:  PR[GP1:91,1] = PR[GP1:90,1] + 93.549;
   1:  PR[GP1:91,2] = PR[GP1:90,2] + 92.006;
   1:L PR[91] 10mm/sec FINE;
   1:  PR[GP1:91,1] = PR[GP1:90,1] + 94.110;
   1:  PR[GP1:91,2] = PR[GP1:90,2] + 92.247;
   1:L PR[91] 10mm/sec FINE;
   1:  PR[GP1:91,1] = PR[GP1:90,1] + 95.158;
   1:  PR[GP1:91,2] = PR[GP1:90,2] + 92.759;
   1:L PR[91] 10mm/sec FINE;
   1:  PR[GP1:91,1] = PR[GP1:90,1] + 96.004;
   1:  PR[GP1:91,2] = PR[GP1:90,2] + 92.966;
   1:L PR[91] 10mm/sec FINE;
   1:  PR[GP1:91,1] = PR[GP1:90,1] + 97.189;
   1:  PR[GP1:91,2] = PR[GP1:90,2] + 92.599;
   1:L PR[91] 10mm/sec FINE;
   1:  PR[GP1:91,1] = PR[GP1:90,1] + 99.678;
   1:  PR[GP1:91,2] = PR[GP1:90,2] + 91.289;
   1:L PR[91] 10mm/sec FINE;
   1:  PR[GP1:91,1] = PR[GP1:90,1] + 102.309;
   1:  PR[GP1:91,2] = PR[GP1:90,2] + 90.398;
   1:L PR[91] 10mm/sec FINE;
   1:  PR[GP1:91,1] = PR[GP1:90,1] + 102.826;
   1:  PR[GP1:91,2] = PR[GP1:90,2] + 90.288;
   1:L PR[91] 10mm/sec FINE;
   1:  PR[GP1:91,1] = PR[GP1:90,1] + 105.003;
   1:  PR[GP1:91,2] = PR[GP1:90,2] + 89.924;
   1:L PR[91] 10mm/sec FINE;
   1:  PR[GP1:91,1] = PR[GP1:90,1] + 106.001;
   1:  PR[GP1:91,2] = PR[GP1:90,2] + 89.865;
   1:L PR[91] 10mm/sec FINE;
   1:  PR[GP1:91,1] = PR[GP1:90,1] + 107.680;
   1:  PR[GP1:91,2] = PR[GP1:90,2] + 89.848;
   1:L PR[91] 10mm/sec FINE;
   1:  PR[GP1:91,1] = PR[GP1:90,1] + 109.271;
   1:  PR[GP1:91,2] = PR[GP1:90,2] + 89.989;
   1:L PR[91] 10mm/sec FINE;
   1:  PR[GP1:91,1] = PR[GP1:90,1] + 110.263;
   1:  PR[GP1:91,2] = PR[GP1:90,2] + 90.131;
   1:L PR[91] 10mm/sec FINE;
   1:  PR[GP1:91,1] = PR[GP1:90,1] + 112.508;
   1:  PR[GP1:91,2] = PR[GP1:90,2] + 90.665;
   1:L PR[91] 10mm/sec FINE;
   1:  PR[GP1:91,1] = PR[GP1:90,1] + 112.695;
   1:  PR[GP1:91,2] = PR[GP1:90,2] + 90.722;
   1:L PR[91] 10mm/sec FINE;
   1:  PR[GP1:91,1] = PR[GP1:90,1] + 113.241;
   1:  PR[GP1:91,2] = PR[GP1:90,2] + 90.938;
   1:L PR[91] 10mm/sec FINE;
   1:  PR[GP1:91,1] = PR[GP1:90,1] + 115.234;
   1:  PR[GP1:91,2] = PR[GP1:90,2] + 91.663;
   1:L PR[91] 10mm/sec FINE;
   1:  PR[GP1:91,1] = PR[GP1:90,1] + 117.703;
   1:  PR[GP1:91,2] = PR[GP1:90,2] + 92.961;
   1:L PR[91] 10mm/sec FINE;
   1:  PR[GP1:91,1] = PR[GP1:90,1] + 119.984;
   1:  PR[GP1:91,2] = PR[GP1:90,2] + 94.586;
   1:L PR[91] 10mm/sec FINE;
   1:  PR[GP1:91,1] = PR[GP1:90,1] + 121.266;
   1:  PR[GP1:91,2] = PR[GP1:90,2] + 95.801;
   1:L PR[91] 10mm/sec FINE;
   1:  PR[GP1:91,1] = PR[GP1:90,1] + 122.042;
   1:  PR[GP1:91,2] = PR[GP1:90,2] + 96.502;
   1:L PR[91] 10mm/sec FINE;
   1:  PR[GP1:91,1] = PR[GP1:90,1] + 123.829;
   1:  PR[GP1:91,2] = PR[GP1:90,2] + 98.659;
   1:L PR[91] 10mm/sec FINE;
   1:  PR[GP1:91,1] = PR[GP1:90,1] + 125.278;
   1:  PR[GP1:91,2] = PR[GP1:90,2] + 101.046;
   1:L PR[91] 10mm/sec FINE;
   1:  PR[GP1:91,1] = PR[GP1:90,1] + 126.061;
   1:  PR[GP1:91,2] = PR[GP1:90,2] + 102.913;
   1:L PR[91] 10mm/sec FINE;
   1:  PR[GP1:91,1] = PR[GP1:90,1] + 126.346;
   1:  PR[GP1:91,2] = PR[GP1:90,2] + 103.608;
   1:L PR[91] 10mm/sec FINE;
   1:  PR[GP1:91,1] = PR[GP1:90,1] + 126.997;
   1:  PR[GP1:91,2] = PR[GP1:90,2] + 106.286;
   1:L PR[91] 10mm/sec FINE;
   1:  PR[GP1:91,1] = PR[GP1:90,1] + 127.192;
   1:  PR[GP1:91,2] = PR[GP1:90,2] + 109.013;
   1:L PR[91] 10mm/sec FINE;
   1:  PR[GP1:91,1] = PR[GP1:90,1] + 126.796;
   1:  PR[GP1:91,2] = PR[GP1:90,2] + 112.454;
   1:L PR[91] 10mm/sec FINE;
   1:  PR[GP1:91,1] = PR[GP1:90,1] + 125.677;
   1:  PR[GP1:91,2] = PR[GP1:90,2] + 115.738;
   1:L PR[91] 10mm/sec FINE;
   1:  PR[GP1:91,1] = PR[GP1:90,1] + 123.869;
   1:  PR[GP1:91,2] = PR[GP1:90,2] + 118.725;
   1:L PR[91] 10mm/sec FINE;
   1:  PR[GP1:91,1] = PR[GP1:90,1] + 121.447;
   1:  PR[GP1:91,2] = PR[GP1:90,2] + 121.305;
   1:L PR[91] 10mm/sec FINE;
   1:  PR[GP1:91,1] = PR[GP1:90,1] + 118.507;
   1:  PR[GP1:91,2] = PR[GP1:90,2] + 123.382;
   1:L PR[91] 10mm/sec FINE;
   1:  PR[GP1:91,1] = PR[GP1:90,1] + 115.210;
   1:  PR[GP1:91,2] = PR[GP1:90,2] + 124.846;
   1:L PR[91] 10mm/sec FINE;
   1:  PR[GP1:91,1] = PR[GP1:90,1] + 111.633;
   1:  PR[GP1:91,2] = PR[GP1:90,2] + 125.680;
   1:L PR[91] 10mm/sec FINE;
   1:  PR[GP1:91,1] = PR[GP1:90,1] + 110.939;
   1:  PR[GP1:91,2] = PR[GP1:90,2] + 125.713;
   1:L PR[91] 10mm/sec FINE;
   1:  PR[GP1:91,1] = PR[GP1:90,1] + 107.952;
   1:  PR[GP1:91,2] = PR[GP1:90,2] + 125.838;
   1:L PR[91] 10mm/sec FINE;
   1:  PR[GP1:91,1] = PR[GP1:90,1] + 106.900;
   1:  PR[GP1:91,2] = PR[GP1:90,2] + 125.698;
   1:L PR[91] 10mm/sec FINE;
   1:  PR[GP1:91,1] = PR[GP1:90,1] + 104.320;
   1:  PR[GP1:91,2] = PR[GP1:90,2] + 125.317;
   1:L PR[91] 10mm/sec FINE;
   1:  PR[GP1:91,1] = PR[GP1:90,1] + 100.826;
   1:  PR[GP1:91,2] = PR[GP1:90,2] + 124.150;
   1:L PR[91] 10mm/sec FINE;
   1:  PR[GP1:91,1] = PR[GP1:90,1] + 99.347;
   1:  PR[GP1:91,2] = PR[GP1:90,2] + 123.352;
   1:L PR[91] 10mm/sec FINE;
   1:  PR[GP1:91,1] = PR[GP1:90,1] + 97.636;
   1:  PR[GP1:91,2] = PR[GP1:90,2] + 122.376;
   1:L PR[91] 10mm/sec FINE;
   1:  PR[GP1:91,1] = PR[GP1:90,1] + 97.505;
   1:  PR[GP1:91,2] = PR[GP1:90,2] + 122.294;
   1:L PR[91] 10mm/sec FINE;
   1:  PR[GP1:91,1] = PR[GP1:90,1] + 96.348;
   1:  PR[GP1:91,2] = PR[GP1:90,2] + 121.426;
   1:L PR[91] 10mm/sec FINE;
   1:  PR[GP1:91,1] = PR[GP1:90,1] + 96.058;
   1:  PR[GP1:91,2] = PR[GP1:90,2] + 121.307;
   1:L PR[91] 10mm/sec FINE;
   1:  PR[GP1:91,1] = PR[GP1:90,1] + 95.434;
   1:  PR[GP1:91,2] = PR[GP1:90,2] + 120.964;
   1:L PR[91] 10mm/sec FINE;
   1:  PR[GP1:91,1] = PR[GP1:90,1] + 95.313;
   1:  PR[GP1:91,2] = PR[GP1:90,2] + 120.950;
   1:L PR[91] 10mm/sec FINE;
   1:  PR[GP1:91,1] = PR[GP1:90,1] + 94.949;
   1:  PR[GP1:91,2] = PR[GP1:90,2] + 121.001;
   1:L PR[91] 10mm/sec FINE;
   1:  PR[GP1:91,1] = PR[GP1:90,1] + 94.346;
   1:  PR[GP1:91,2] = PR[GP1:90,2] + 121.012;
   1:L PR[91] 10mm/sec FINE;
   1:  PR[GP1:91,1] = PR[GP1:90,1] + 93.789;
   1:  PR[GP1:91,2] = PR[GP1:90,2] + 121.310;
   1:L PR[91] 10mm/sec FINE;
   1:  PR[GP1:91,1] = PR[GP1:90,1] + 91.707;
   1:  PR[GP1:91,2] = PR[GP1:90,2] + 122.568;
   1:L PR[91] 10mm/sec FINE;
   1:  PR[GP1:91,1] = PR[GP1:90,1] + 91.384;
   1:  PR[GP1:91,2] = PR[GP1:90,2] + 122.727;
   1:L PR[91] 10mm/sec FINE;
   1:  PR[GP1:91,1] = PR[GP1:90,1] + 90.557;
   1:  PR[GP1:91,2] = PR[GP1:90,2] + 123.067;
   1:L PR[91] 10mm/sec FINE;
   1:  PR[GP1:91,1] = PR[GP1:90,1] + 88.541;
   1:  PR[GP1:91,2] = PR[GP1:90,2] + 123.985;
   1:L PR[91] 10mm/sec FINE;
   1:  PR[GP1:91,1] = PR[GP1:90,1] + 87.338;
   1:  PR[GP1:91,2] = PR[GP1:90,2] + 124.428;
   1:L PR[91] 10mm/sec FINE;
   1:  PR[GP1:91,1] = PR[GP1:90,1] + 85.481;
   1:  PR[GP1:91,2] = PR[GP1:90,2] + 124.923;
   1:L PR[91] 10mm/sec FINE;
   1:  PR[GP1:91,1] = PR[GP1:90,1] + 82.554;
   1:  PR[GP1:91,2] = PR[GP1:90,2] + 125.441;
   1:L PR[91] 10mm/sec FINE;
   1:  PR[GP1:91,1] = PR[GP1:90,1] + 82.103;
   1:  PR[GP1:91,2] = PR[GP1:90,2] + 125.483;
   1:L PR[91] 10mm/sec FINE;
   1:  PR[GP1:91,1] = PR[GP1:90,1] + 78.839;
   1:  PR[GP1:91,2] = PR[GP1:90,2] + 125.469;
   1:L PR[91] 10mm/sec FINE;
   1:  PR[GP1:91,1] = PR[GP1:90,1] + 78.230;
   1:  PR[GP1:91,2] = PR[GP1:90,2] + 125.449;
   1:L PR[91] 10mm/sec FINE;
   1:  PR[GP1:91,1] = PR[GP1:90,1] + 75.756;
   1:  PR[GP1:91,2] = PR[GP1:90,2] + 124.948;
   1:L PR[91] 10mm/sec FINE;
   1:  PR[GP1:91,1] = PR[GP1:90,1] + 74.389;
   1:  PR[GP1:91,2] = PR[GP1:90,2] + 124.638;
   1:L PR[91] 10mm/sec FINE;
   1:  PR[GP1:91,1] = PR[GP1:90,1] + 72.740;
   1:  PR[GP1:91,2] = PR[GP1:90,2] + 123.943;
   1:L PR[91] 10mm/sec FINE;
   1:  PR[GP1:91,1] = PR[GP1:90,1] + 70.901;
   1:  PR[GP1:91,2] = PR[GP1:90,2] + 123.124;
   1:L PR[91] 10mm/sec FINE;
   1:  PR[GP1:91,1] = PR[GP1:90,1] + 69.895;
   1:  PR[GP1:91,2] = PR[GP1:90,2] + 122.426;
   1:L PR[91] 10mm/sec FINE;
   1:  PR[GP1:91,1] = PR[GP1:90,1] + 67.890;
   1:  PR[GP1:91,2] = PR[GP1:90,2] + 120.990;
   1:L PR[91] 10mm/sec FINE;
   1:  PR[GP1:91,1] = PR[GP1:90,1] + 65.467;
   1:  PR[GP1:91,2] = PR[GP1:90,2] + 118.327;
   1:L PR[91] 10mm/sec FINE;
   1:  PR[GP1:91,1] = PR[GP1:90,1] + 63.700;
   1:  PR[GP1:91,2] = PR[GP1:90,2] + 115.252;
   1:L PR[91] 10mm/sec FINE;
   1:  PR[GP1:91,1] = PR[GP1:90,1] + 62.624;
   1:  PR[GP1:91,2] = PR[GP1:90,2] + 111.901;
   1:L PR[91] 10mm/sec FINE;
   1:  PR[GP1:91,1] = PR[GP1:90,1] + 62.372;
   1:  PR[GP1:91,2] = PR[GP1:90,2] + 108.357;
   1:L PR[91] 10mm/sec FINE;
   1:  PR[GP1:91,1] = PR[GP1:90,1] + 62.912;
   1:  PR[GP1:91,2] = PR[GP1:90,2] + 104.750;
   1:L PR[91] 10mm/sec FINE;
   1:  PR[GP1:91,1] = PR[GP1:90,1] + 64.182;
   1:  PR[GP1:91,2] = PR[GP1:90,2] + 101.278;
   1:L PR[91] 10mm/sec FINE;
   1:  PR[GP1:91,1] = PR[GP1:90,1] + 65.295;
   1:  PR[GP1:91,2] = PR[GP1:90,2] + 99.500;
   1:L PR[91] 10mm/sec FINE;
   1:  PR[GP1:91,1] = PR[GP1:90,1] + 66.256;
   1:  PR[GP1:91,2] = PR[GP1:90,2] + 98.038;
   1:L PR[91] 10mm/sec FINE;
   1:  PR[GP1:91,1] = PR[GP1:90,1] + 67.294;
   1:  PR[GP1:91,2] = PR[GP1:90,2] + 96.943;
   1:L PR[91] 10mm/sec FINE;
   1:  PR[GP1:91,1] = PR[GP1:90,1] + 69.056;
   1:  PR[GP1:91,2] = PR[GP1:90,2] + 95.185;
   1:L PR[91] 10mm/sec FINE;
   1:  PR[GP1:91,1] = PR[GP1:90,1] + 69.649;
   1:  PR[GP1:91,2] = PR[GP1:90,2] + 94.762;
   1:L PR[91] 10mm/sec FINE;
   1:  PR[GP1:91,1] = PR[GP1:90,1] + 70.077;
   1:  PR[GP1:91,2] = PR[GP1:90,2] + 94.638;
   1:  PR[GP1:91,3] = PR[GP1:90,3] + 27.900;
   1:L PR[91] 10mm/sec FINE;
   1:  PR[GP1:91,1] = PR[GP1:90,1] + 72.862;
   1:  PR[GP1:91,2] = PR[GP1:90,2] + 92.824;
   1:L PR[91] 10mm/sec FINE;
   1:  PR[GP1:91,1] = PR[GP1:90,1] + 74.143;
   1:  PR[GP1:91,2] = PR[GP1:90,2] + 92.237;
   1:L PR[91] 10mm/sec FINE;
   1:  PR[GP1:91,1] = PR[GP1:90,1] + 76.360;
   1:  PR[GP1:91,2] = PR[GP1:90,2] + 91.313;
   1:L PR[91] 10mm/sec FINE;
   1:  PR[GP1:91,1] = PR[GP1:90,1] + 79.633;
   1:  PR[GP1:91,2] = PR[GP1:90,2] + 90.455;
   1:L PR[91] 10mm/sec FINE;
   1:  PR[GP1:91,1] = PR[GP1:90,1] + 79.869;
   1:  PR[GP1:91,2] = PR[GP1:90,2] + 90.403;
   1:L PR[91] 10mm/sec FINE;
   1:  PR[GP1:91,1] = PR[GP1:90,1] + 83.230;
   1:  PR[GP1:91,2] = PR[GP1:90,2] + 90.041;
   1:L PR[91] 10mm/sec FINE;
   1:  PR[GP1:91,1] = PR[GP1:90,1] + 84.482;
   1:  PR[GP1:91,2] = PR[GP1:90,2] + 89.972;
   1:L PR[91] 10mm/sec FINE;
   1:  PR[GP1:91,1] = PR[GP1:90,1] + 86.033;
   1:  PR[GP1:91,2] = PR[GP1:90,2] + 90.061;
   1:L PR[91] 10mm/sec FINE;
   1:  PR[GP1:91,1] = PR[GP1:90,1] + 88.285;
   1:  PR[GP1:91,2] = PR[GP1:90,2] + 90.221;
   1:L PR[91] 10mm/sec FINE;
   1:  PR[GP1:91,1] = PR[GP1:90,1] + 91.708;
   1:  PR[GP1:91,2] = PR[GP1:90,2] + 90.831;
   1:L PR[91] 10mm/sec FINE;
   1:  PR[GP1:91,1] = PR[GP1:90,1] + 94.203;
   1:  PR[GP1:91,2] = PR[GP1:90,2] + 91.667;
   1:L PR[91] 10mm/sec FINE;
   1:  PR[GP1:91,1] = PR[GP1:90,1] + 94.544;
   1:  PR[GP1:91,2] = PR[GP1:90,2] + 91.807;
   1:L PR[91] 10mm/sec FINE;
   1:  PR[GP1:91,1] = PR[GP1:90,1] + 95.464;
   1:  PR[GP1:91,2] = PR[GP1:90,2] + 92.236;
   1:L PR[91] 10mm/sec FINE;
   1:  PR[GP1:91,1] = PR[GP1:90,1] + 96.205;
   1:  PR[GP1:91,2] = PR[GP1:90,2] + 92.411;
   1:L PR[91] 10mm/sec FINE;
   1:  PR[GP1:91,1] = PR[GP1:90,1] + 97.401;
   1:  PR[GP1:91,2] = PR[GP1:90,2] + 92.091;
   1:L PR[91] 10mm/sec FINE;
   1:  PR[GP1:91,1] = PR[GP1:90,1] + 99.137;
   1:  PR[GP1:91,2] = PR[GP1:90,2] + 91.199;
   1:L PR[91] 10mm/sec FINE;
   1:  PR[GP1:91,1] = PR[GP1:90,1] + 99.452;
   1:  PR[GP1:91,2] = PR[GP1:90,2] + 91.053;
   1:L PR[91] 10mm/sec FINE;
   1:  PR[GP1:91,1] = PR[GP1:90,1] + 102.151;
   1:  PR[GP1:91,2] = PR[GP1:90,2] + 90.145;
   1:L PR[91] 10mm/sec FINE;
   1:  PR[GP1:91,1] = PR[GP1:90,1] + 104.933;
   1:  PR[GP1:91,2] = PR[GP1:90,2] + 89.686;
   1:L PR[91] 10mm/sec FINE;
   1:  PR[GP1:91,1] = PR[GP1:90,1] + 105.175;
   1:  PR[GP1:91,2] = PR[GP1:90,2] + 89.671;
   1:L PR[91] 10mm/sec FINE;
   1:  PR[GP1:91,1] = PR[GP1:90,1] + 107.664;
   1:  PR[GP1:91,2] = PR[GP1:90,2] + 89.646;
   1:L PR[91] 10mm/sec FINE;
   1:  PR[GP1:91,1] = PR[GP1:90,1] + 108.458;
   1:  PR[GP1:91,2] = PR[GP1:90,2] + 89.717;
   1:L PR[91] 10mm/sec FINE;
   1:  PR[GP1:91,1] = PR[GP1:90,1] + 110.297;
   1:  PR[GP1:91,2] = PR[GP1:90,2] + 89.981;
   1:L PR[91] 10mm/sec FINE;
   1:  PR[GP1:91,1] = PR[GP1:90,1] + 111.727;
   1:  PR[GP1:91,2] = PR[GP1:90,2] + 90.321;
   1:L PR[91] 10mm/sec FINE;
   1:  PR[GP1:91,1] = PR[GP1:90,1] + 112.772;
   1:  PR[GP1:91,2] = PR[GP1:90,2] + 90.638;
   1:L PR[91] 10mm/sec FINE;
   1:  PR[GP1:91,1] = PR[GP1:90,1] + 114.850;
   1:  PR[GP1:91,2] = PR[GP1:90,2] + 91.461;
   1:L PR[91] 10mm/sec FINE;
   1:  PR[GP1:91,1] = PR[GP1:90,1] + 115.051;
   1:  PR[GP1:91,2] = PR[GP1:90,2] + 91.557;
   1:L PR[91] 10mm/sec FINE;
   1:  PR[GP1:91,1] = PR[GP1:90,1] + 115.594;
   1:  PR[GP1:91,2] = PR[GP1:90,2] + 91.866;
   1:L PR[91] 10mm/sec FINE;
   1:  PR[GP1:91,1] = PR[GP1:90,1] + 117.422;
   1:  PR[GP1:91,2] = PR[GP1:90,2] + 92.836;
   1:L PR[91] 10mm/sec FINE;
   1:  PR[GP1:91,1] = PR[GP1:90,1] + 119.689;
   1:  PR[GP1:91,2] = PR[GP1:90,2] + 94.467;
   1:L PR[91] 10mm/sec FINE;
   1:  PR[GP1:91,1] = PR[GP1:90,1] + 121.174;
   1:  PR[GP1:91,2] = PR[GP1:90,2] + 95.876;
   1:L PR[91] 10mm/sec FINE;
   1:  PR[GP1:91,1] = PR[GP1:90,1] + 121.712;
   1:  PR[GP1:91,2] = PR[GP1:90,2] + 96.396;
   1:L PR[91] 10mm/sec FINE;
   1:  PR[GP1:91,1] = PR[GP1:90,1] + 122.925;
   1:  PR[GP1:91,2] = PR[GP1:90,2] + 97.936;
   1:L PR[91] 10mm/sec FINE;
   1:  PR[GP1:91,1] = PR[GP1:90,1] + 123.459;
   1:  PR[GP1:91,2] = PR[GP1:90,2] + 98.582;
   1:L PR[91] 10mm/sec FINE;
   1:  PR[GP1:91,1] = PR[GP1:90,1] + 124.892;
   1:  PR[GP1:91,2] = PR[GP1:90,2] + 100.963;
   1:L PR[91] 10mm/sec FINE;
   1:  PR[GP1:91,1] = PR[GP1:90,1] + 125.294;
   1:  PR[GP1:91,2] = PR[GP1:90,2] + 101.920;
   1:L PR[91] 10mm/sec FINE;
   1:  PR[GP1:91,1] = PR[GP1:90,1] + 125.949;
   1:  PR[GP1:91,2] = PR[GP1:90,2] + 103.515;
   1:L PR[91] 10mm/sec FINE;
   1:  PR[GP1:91,1] = PR[GP1:90,1] + 126.592;
   1:  PR[GP1:91,2] = PR[GP1:90,2] + 106.180;
   1:L PR[91] 10mm/sec FINE;
   1:  PR[GP1:91,1] = PR[GP1:90,1] + 126.773;
   1:  PR[GP1:91,2] = PR[GP1:90,2] + 108.906;
   1:L PR[91] 10mm/sec FINE;
   1:  PR[GP1:91,1] = PR[GP1:90,1] + 126.371;
   1:  PR[GP1:91,2] = PR[GP1:90,2] + 112.360;
   1:L PR[91] 10mm/sec FINE;
   1:  PR[GP1:91,1] = PR[GP1:90,1] + 125.250;
   1:  PR[GP1:91,2] = PR[GP1:90,2] + 115.646;
   1:L PR[91] 10mm/sec FINE;
   1:  PR[GP1:91,1] = PR[GP1:90,1] + 123.438;
   1:  PR[GP1:91,2] = PR[GP1:90,2] + 118.636;
   1:L PR[91] 10mm/sec FINE;
   1:  PR[GP1:91,1] = PR[GP1:90,1] + 121.011;
   1:  PR[GP1:91,2] = PR[GP1:90,2] + 121.218;
   1:L PR[91] 10mm/sec FINE;
   1:  PR[GP1:91,1] = PR[GP1:90,1] + 118.105;
   1:  PR[GP1:91,2] = PR[GP1:90,2] + 123.270;
   1:L PR[91] 10mm/sec FINE;
   1:  PR[GP1:91,1] = PR[GP1:90,1] + 114.808;
   1:  PR[GP1:91,2] = PR[GP1:90,2] + 124.734;
   1:L PR[91] 10mm/sec FINE;
   1:  PR[GP1:91,1] = PR[GP1:90,1] + 111.230;
   1:  PR[GP1:91,2] = PR[GP1:90,2] + 125.570;
   1:L PR[91] 10mm/sec FINE;
   1:  PR[GP1:91,1] = PR[GP1:90,1] + 107.568;
   1:  PR[GP1:91,2] = PR[GP1:90,2] + 125.721;
   1:L PR[91] 10mm/sec FINE;
   1:  PR[GP1:91,1] = PR[GP1:90,1] + 103.960;
   1:  PR[GP1:91,2] = PR[GP1:90,2] + 125.192;
   1:L PR[91] 10mm/sec FINE;
   1:  PR[GP1:91,1] = PR[GP1:90,1] + 100.468;
   1:  PR[GP1:91,2] = PR[GP1:90,2] + 124.028;
   1:L PR[91] 10mm/sec FINE;
   1:  PR[GP1:91,1] = PR[GP1:90,1] + 97.324;
   1:  PR[GP1:91,2] = PR[GP1:90,2] + 122.248;
   1:L PR[91] 10mm/sec FINE;
   1:  PR[GP1:91,1] = PR[GP1:90,1] + 97.110;
   1:  PR[GP1:91,2] = PR[GP1:90,2] + 122.114;
   1:L PR[91] 10mm/sec FINE;
   1:  PR[GP1:91,1] = PR[GP1:90,1] + 96.454;
   1:  PR[GP1:91,2] = PR[GP1:90,2] + 121.622;
   1:L PR[91] 10mm/sec FINE;
   1:  PR[GP1:91,1] = PR[GP1:90,1] + 95.908;
   1:  PR[GP1:91,2] = PR[GP1:90,2] + 121.398;
   1:L PR[91] 10mm/sec FINE;
   1:  PR[GP1:91,1] = PR[GP1:90,1] + 95.525;
   1:  PR[GP1:91,2] = PR[GP1:90,2] + 121.188;
   1:L PR[91] 10mm/sec FINE;
   1:  PR[GP1:91,1] = PR[GP1:90,1] + 95.375;
   1:  PR[GP1:91,2] = PR[GP1:90,2] + 121.170;
   1:L PR[91] 10mm/sec FINE;
   1:  PR[GP1:91,1] = PR[GP1:90,1] + 94.825;
   1:  PR[GP1:91,2] = PR[GP1:90,2] + 121.247;
   1:L PR[91] 10mm/sec FINE;
   1:  PR[GP1:91,1] = PR[GP1:90,1] + 94.440;
   1:  PR[GP1:91,2] = PR[GP1:90,2] + 121.254;
   1:L PR[91] 10mm/sec FINE;
   1:  PR[GP1:91,1] = PR[GP1:90,1] + 93.987;
   1:  PR[GP1:91,2] = PR[GP1:90,2] + 121.489;
   1:L PR[91] 10mm/sec FINE;
   1:  PR[GP1:91,1] = PR[GP1:90,1] + 92.694;
   1:  PR[GP1:91,2] = PR[GP1:90,2] + 122.270;
   1:L PR[91] 10mm/sec FINE;
   1:  PR[GP1:91,1] = PR[GP1:90,1] + 91.701;
   1:  PR[GP1:91,2] = PR[GP1:90,2] + 122.758;
   1:L PR[91] 10mm/sec FINE;
   1:  PR[GP1:91,1] = PR[GP1:90,1] + 89.227;
   1:  PR[GP1:91,2] = PR[GP1:90,2] + 123.774;
   1:L PR[91] 10mm/sec FINE;
   1:  PR[GP1:91,1] = PR[GP1:90,1] + 88.657;
   1:  PR[GP1:91,2] = PR[GP1:90,2] + 124.034;
   1:L PR[91] 10mm/sec FINE;
   1:  PR[GP1:91,1] = PR[GP1:90,1] + 88.326;
   1:  PR[GP1:91,2] = PR[GP1:90,2] + 124.156;
   1:L PR[91] 10mm/sec FINE;
   1:  PR[GP1:91,1] = PR[GP1:90,1] + 85.632;
   1:  PR[GP1:91,2] = PR[GP1:90,2] + 124.874;
   1:L PR[91] 10mm/sec FINE;
   1:  PR[GP1:91,1] = PR[GP1:90,1] + 83.588;
   1:  PR[GP1:91,2] = PR[GP1:90,2] + 125.236;
   1:L PR[91] 10mm/sec FINE;
   1:  PR[GP1:91,1] = PR[GP1:90,1] + 82.304;
   1:  PR[GP1:91,2] = PR[GP1:90,2] + 125.355;
   1:L PR[91] 10mm/sec FINE;
   1:  PR[GP1:91,1] = PR[GP1:90,1] + 78.741;
   1:  PR[GP1:91,2] = PR[GP1:90,2] + 125.341;
   1:L PR[91] 10mm/sec FINE;
   1:  PR[GP1:91,1] = PR[GP1:90,1] + 75.692;
   1:  PR[GP1:91,2] = PR[GP1:90,2] + 124.725;
   1:L PR[91] 10mm/sec FINE;
   1:  PR[GP1:91,1] = PR[GP1:90,1] + 74.878;
   1:  PR[GP1:91,2] = PR[GP1:90,2] + 124.540;
   1:L PR[91] 10mm/sec FINE;
   1:  PR[GP1:91,1] = PR[GP1:90,1] + 72.715;
   1:  PR[GP1:91,2] = PR[GP1:90,2] + 123.627;
   1:L PR[91] 10mm/sec FINE;
   1:  PR[GP1:91,1] = PR[GP1:90,1] + 71.368;
   1:  PR[GP1:91,2] = PR[GP1:90,2] + 123.028;
   1:L PR[91] 10mm/sec FINE;
   1:  PR[GP1:91,1] = PR[GP1:90,1] + 69.922;
   1:  PR[GP1:91,2] = PR[GP1:90,2] + 122.025;
   1:L PR[91] 10mm/sec FINE;
   1:  PR[GP1:91,1] = PR[GP1:90,1] + 68.340;
   1:  PR[GP1:91,2] = PR[GP1:90,2] + 120.891;
   1:L PR[91] 10mm/sec FINE;
   1:  PR[GP1:91,1] = PR[GP1:90,1] + 65.903;
   1:  PR[GP1:91,2] = PR[GP1:90,2] + 118.221;
   1:L PR[91] 10mm/sec FINE;
   1:  PR[GP1:91,1] = PR[GP1:90,1] + 64.128;
   1:  PR[GP1:91,2] = PR[GP1:90,2] + 115.135;
   1:L PR[91] 10mm/sec FINE;
   1:  PR[GP1:91,1] = PR[GP1:90,1] + 63.046;
   1:  PR[GP1:91,2] = PR[GP1:90,2] + 111.774;
   1:L PR[91] 10mm/sec FINE;
   1:  PR[GP1:91,1] = PR[GP1:90,1] + 62.796;
   1:  PR[GP1:91,2] = PR[GP1:90,2] + 108.216;
   1:L PR[91] 10mm/sec FINE;
   1:  PR[GP1:91,1] = PR[GP1:90,1] + 63.135;
   1:  PR[GP1:91,2] = PR[GP1:90,2] + 105.910;
   1:L PR[91] 10mm/sec FINE;
   1:  PR[GP1:91,1] = PR[GP1:90,1] + 63.345;
   1:  PR[GP1:91,2] = PR[GP1:90,2] + 104.592;
   1:L PR[91] 10mm/sec FINE;
   1:  PR[GP1:91,1] = PR[GP1:90,1] + 64.026;
   1:  PR[GP1:91,2] = PR[GP1:90,2] + 102.709;
   1:L PR[91] 10mm/sec FINE;
   1:  PR[GP1:91,1] = PR[GP1:90,1] + 64.627;
   1:  PR[GP1:91,2] = PR[GP1:90,2] + 101.107;
   1:L PR[91] 10mm/sec FINE;
   1:  PR[GP1:91,1] = PR[GP1:90,1] + 65.458;
   1:  PR[GP1:91,2] = PR[GP1:90,2] + 99.780;
   1:L PR[91] 10mm/sec FINE;
   1:  PR[GP1:91,1] = PR[GP1:90,1] + 66.724;
   1:  PR[GP1:91,2] = PR[GP1:90,2] + 97.853;
   1:L PR[91] 10mm/sec FINE;
   1:  PR[GP1:91,1] = PR[GP1:90,1] + 67.376;
   1:  PR[GP1:91,2] = PR[GP1:90,2] + 97.165;
   1:L PR[91] 10mm/sec FINE;
   1:  PR[GP1:91,1] = PR[GP1:90,1] + 69.552;
   1:  PR[GP1:91,2] = PR[GP1:90,2] + 94.993;
   1:L PR[91] 10mm/sec FINE;
   1:  PR[GP1:91,1] = PR[GP1:90,1] + 70.608;
   1:  PR[GP1:91,2] = PR[GP1:90,2] + 94.476;
   1:  PR[GP1:91,3] = PR[GP1:90,3] + 28.900;
   1:L PR[91] 10mm/sec FINE;
   1:  PR[GP1:91,1] = PR[GP1:90,1] + 73.278;
   1:  PR[GP1:91,2] = PR[GP1:90,2] + 92.736;
   1:L PR[91] 10mm/sec FINE;
   1:  PR[GP1:91,1] = PR[GP1:90,1] + 75.510;
   1:  PR[GP1:91,2] = PR[GP1:90,2] + 91.715;
   1:L PR[91] 10mm/sec FINE;
   1:  PR[GP1:91,1] = PR[GP1:90,1] + 76.715;
   1:  PR[GP1:91,2] = PR[GP1:90,2] + 91.213;
   1:L PR[91] 10mm/sec FINE;
   1:  PR[GP1:91,1] = PR[GP1:90,1] + 78.846;
   1:  PR[GP1:91,2] = PR[GP1:90,2] + 90.654;
   1:L PR[91] 10mm/sec FINE;
   1:  PR[GP1:91,1] = PR[GP1:90,1] + 80.236;
   1:  PR[GP1:91,2] = PR[GP1:90,2] + 90.269;
   1:L PR[91] 10mm/sec FINE;
   1:  PR[GP1:91,1] = PR[GP1:90,1] + 80.877;
   1:  PR[GP1:91,2] = PR[GP1:90,2] + 90.151;
   1:L PR[91] 10mm/sec FINE;
   1:  PR[GP1:91,1] = PR[GP1:90,1] + 83.445;
   1:  PR[GP1:91,2] = PR[GP1:90,2] + 89.866;
   1:L PR[91] 10mm/sec FINE;
   1:  PR[GP1:91,1] = PR[GP1:90,1] + 85.433;
   1:  PR[GP1:91,2] = PR[GP1:90,2] + 89.757;
   1:L PR[91] 10mm/sec FINE;
   1:  PR[GP1:91,1] = PR[GP1:90,1] + 87.159;
   1:  PR[GP1:91,2] = PR[GP1:90,2] + 89.870;
   1:L PR[91] 10mm/sec FINE;
   1:  PR[GP1:91,1] = PR[GP1:90,1] + 88.958;
   1:  PR[GP1:91,2] = PR[GP1:90,2] + 89.936;
   1:L PR[91] 10mm/sec FINE;
   1:  PR[GP1:91,1] = PR[GP1:90,1] + 89.525;
   1:  PR[GP1:91,2] = PR[GP1:90,2] + 90.017;
   1:L PR[91] 10mm/sec FINE;
   1:  PR[GP1:91,1] = PR[GP1:90,1] + 92.551;
   1:  PR[GP1:91,2] = PR[GP1:90,2] + 90.551;
   1:L PR[91] 10mm/sec FINE;
   1:  PR[GP1:91,1] = PR[GP1:90,1] + 94.661;
   1:  PR[GP1:91,2] = PR[GP1:90,2] + 91.254;
   1:L PR[91] 10mm/sec FINE;
   1:  PR[GP1:91,1] = PR[GP1:90,1] + 95.275;
   1:  PR[GP1:91,2] = PR[GP1:90,2] + 91.501;
   1:L PR[91] 10mm/sec FINE;
   1:  PR[GP1:91,1] = PR[GP1:90,1] + 95.778;
   1:  PR[GP1:91,2] = PR[GP1:90,2] + 91.729;
   1:L PR[91] 10mm/sec FINE;
   1:  PR[GP1:91,1] = PR[GP1:90,1] + 96.426;
   1:  PR[GP1:91,2] = PR[GP1:90,2] + 91.886;
   1:L PR[91] 10mm/sec FINE;
   1:  PR[GP1:91,1] = PR[GP1:90,1] + 97.051;
   1:  PR[GP1:91,2] = PR[GP1:90,2] + 91.722;
   1:L PR[91] 10mm/sec FINE;
   1:  PR[GP1:91,1] = PR[GP1:90,1] + 97.624;
   1:  PR[GP1:91,2] = PR[GP1:90,2] + 91.599;
   1:L PR[91] 10mm/sec FINE;
   1:  PR[GP1:91,1] = PR[GP1:90,1] + 98.422;
   1:  PR[GP1:91,2] = PR[GP1:90,2] + 91.195;
   1:L PR[91] 10mm/sec FINE;
   1:  PR[GP1:91,1] = PR[GP1:90,1] + 99.210;
   1:  PR[GP1:91,2] = PR[GP1:90,2] + 90.830;
   1:L PR[91] 10mm/sec FINE;
   1:  PR[GP1:91,1] = PR[GP1:90,1] + 101.904;
   1:  PR[GP1:91,2] = PR[GP1:90,2] + 89.915;
   1:L PR[91] 10mm/sec FINE;
   1:  PR[GP1:91,1] = PR[GP1:90,1] + 104.737;
   1:  PR[GP1:91,2] = PR[GP1:90,2] + 89.447;
   1:L PR[91] 10mm/sec FINE;
   1:  PR[GP1:91,1] = PR[GP1:90,1] + 107.641;
   1:  PR[GP1:91,2] = PR[GP1:90,2] + 89.445;
   1:L PR[91] 10mm/sec FINE;
   1:  PR[GP1:91,1] = PR[GP1:90,1] + 110.332;
   1:  PR[GP1:91,2] = PR[GP1:90,2] + 89.831;
   1:L PR[91] 10mm/sec FINE;
   1:  PR[GP1:91,1] = PR[GP1:90,1] + 110.947;
   1:  PR[GP1:91,2] = PR[GP1:90,2] + 89.978;
   1:L PR[91] 10mm/sec FINE;
   1:  PR[GP1:91,1] = PR[GP1:90,1] + 112.849;
   1:  PR[GP1:91,2] = PR[GP1:90,2] + 90.554;
   1:L PR[91] 10mm/sec FINE;
   1:  PR[GP1:91,1] = PR[GP1:90,1] + 114.121;
   1:  PR[GP1:91,2] = PR[GP1:90,2] + 91.058;
   1:L PR[91] 10mm/sec FINE;
   1:  PR[GP1:91,1] = PR[GP1:90,1] + 115.159;
   1:  PR[GP1:91,2] = PR[GP1:90,2] + 91.551;
   1:L PR[91] 10mm/sec FINE;
   1:  PR[GP1:91,1] = PR[GP1:90,1] + 117.039;
   1:  PR[GP1:91,2] = PR[GP1:90,2] + 92.625;
   1:L PR[91] 10mm/sec FINE;
   1:  PR[GP1:91,1] = PR[GP1:90,1] + 117.240;
   1:  PR[GP1:91,2] = PR[GP1:90,2] + 92.761;
   1:L PR[91] 10mm/sec FINE;
   1:  PR[GP1:91,1] = PR[GP1:90,1] + 117.768;
   1:  PR[GP1:91,2] = PR[GP1:90,2] + 93.171;
   1:L PR[91] 10mm/sec FINE;
   1:  PR[GP1:91,1] = PR[GP1:90,1] + 119.393;
   1:  PR[GP1:91,2] = PR[GP1:90,2] + 94.348;
   1:L PR[91] 10mm/sec FINE;
   1:  PR[GP1:91,1] = PR[GP1:90,1] + 121.402;
   1:  PR[GP1:91,2] = PR[GP1:90,2] + 96.278;
   1:L PR[91] 10mm/sec FINE;
   1:  PR[GP1:91,1] = PR[GP1:90,1] + 123.119;
   1:  PR[GP1:91,2] = PR[GP1:90,2] + 98.469;
   1:L PR[91] 10mm/sec FINE;
   1:  PR[GP1:91,1] = PR[GP1:90,1] + 124.506;
   1:  PR[GP1:91,2] = PR[GP1:90,2] + 100.877;
   1:L PR[91] 10mm/sec FINE;
   1:  PR[GP1:91,1] = PR[GP1:90,1] + 125.552;
   1:  PR[GP1:91,2] = PR[GP1:90,2] + 103.422;
   1:L PR[91] 10mm/sec FINE;
   1:  PR[GP1:91,1] = PR[GP1:90,1] + 126.187;
   1:  PR[GP1:91,2] = PR[GP1:90,2] + 106.075;
   1:L PR[91] 10mm/sec FINE;
   1:  PR[GP1:91,1] = PR[GP1:90,1] + 126.359;
   1:  PR[GP1:91,2] = PR[GP1:90,2] + 108.794;
   1:L PR[91] 10mm/sec FINE;
   1:  PR[GP1:91,1] = PR[GP1:90,1] + 125.947;
   1:  PR[GP1:91,2] = PR[GP1:90,2] + 112.265;
   1:L PR[91] 10mm/sec FINE;
   1:  PR[GP1:91,1] = PR[GP1:90,1] + 124.823;
   1:  PR[GP1:91,2] = PR[GP1:90,2] + 115.554;
   1:L PR[91] 10mm/sec FINE;
   1:  PR[GP1:91,1] = PR[GP1:90,1] + 123.011;
   1:  PR[GP1:91,2] = PR[GP1:90,2] + 118.544;
   1:L PR[91] 10mm/sec FINE;
   1:  PR[GP1:91,1] = PR[GP1:90,1] + 120.612;
   1:  PR[GP1:91,2] = PR[GP1:90,2] + 121.104;
   1:L PR[91] 10mm/sec FINE;
   1:  PR[GP1:91,1] = PR[GP1:90,1] + 117.709;
   1:  PR[GP1:91,2] = PR[GP1:90,2] + 123.153;
   1:L PR[91] 10mm/sec FINE;
   1:  PR[GP1:91,1] = PR[GP1:90,1] + 114.406;
   1:  PR[GP1:91,2] = PR[GP1:90,2] + 124.621;
   1:L PR[91] 10mm/sec FINE;
   1:  PR[GP1:91,1] = PR[GP1:90,1] + 110.879;
   1:  PR[GP1:91,2] = PR[GP1:90,2] + 125.437;
   1:L PR[91] 10mm/sec FINE;
   1:  PR[GP1:91,1] = PR[GP1:90,1] + 108.300;
   1:  PR[GP1:91,2] = PR[GP1:90,2] + 125.544;
   1:L PR[91] 10mm/sec FINE;
   1:  PR[GP1:91,1] = PR[GP1:90,1] + 107.240;
   1:  PR[GP1:91,2] = PR[GP1:90,2] + 125.584;
   1:L PR[91] 10mm/sec FINE;
   1:  PR[GP1:91,1] = PR[GP1:90,1] + 103.601;
   1:  PR[GP1:91,2] = PR[GP1:90,2] + 125.067;
   1:L PR[91] 10mm/sec FINE;
   1:  PR[GP1:91,1] = PR[GP1:90,1] + 102.109;
   1:  PR[GP1:91,2] = PR[GP1:90,2] + 124.570;
   1:L PR[91] 10mm/sec FINE;
   1:  PR[GP1:91,1] = PR[GP1:90,1] + 100.160;
   1:  PR[GP1:91,2] = PR[GP1:90,2] + 123.893;
   1:L PR[91] 10mm/sec FINE;
   1:  PR[GP1:91,1] = PR[GP1:90,1] + 99.001;
   1:  PR[GP1:91,2] = PR[GP1:90,2] + 123.255;
   1:L PR[91] 10mm/sec FINE;
   1:  PR[GP1:91,1] = PR[GP1:90,1] + 97.013;
   1:  PR[GP1:91,2] = PR[GP1:90,2] + 122.121;
   1:L PR[91] 10mm/sec FINE;
   1:  PR[GP1:91,1] = PR[GP1:90,1] + 96.715;
   1:  PR[GP1:91,2] = PR[GP1:90,2] + 121.935;
   1:L PR[91] 10mm/sec FINE;
   1:  PR[GP1:91,1] = PR[GP1:90,1] + 96.560;
   1:  PR[GP1:91,2] = PR[GP1:90,2] + 121.818;
   1:L PR[91] 10mm/sec FINE;
   1:  PR[GP1:91,1] = PR[GP1:90,1] + 95.758;
   1:  PR[GP1:91,2] = PR[GP1:90,2] + 121.490;
   1:L PR[91] 10mm/sec FINE;
   1:  PR[GP1:91,1] = PR[GP1:90,1] + 95.616;
   1:  PR[GP1:91,2] = PR[GP1:90,2] + 121.412;
   1:L PR[91] 10mm/sec FINE;
   1:  PR[GP1:91,1] = PR[GP1:90,1] + 95.436;
   1:  PR[GP1:91,2] = PR[GP1:90,2] + 121.391;
   1:L PR[91] 10mm/sec FINE;
   1:  PR[GP1:91,1] = PR[GP1:90,1] + 94.702;
   1:  PR[GP1:91,2] = PR[GP1:90,2] + 121.494;
   1:L PR[91] 10mm/sec FINE;
   1:  PR[GP1:91,1] = PR[GP1:90,1] + 94.536;
   1:  PR[GP1:91,2] = PR[GP1:90,2] + 121.497;
   1:L PR[91] 10mm/sec FINE;
   1:  PR[GP1:91,1] = PR[GP1:90,1] + 94.185;
   1:  PR[GP1:91,2] = PR[GP1:90,2] + 121.667;
   1:L PR[91] 10mm/sec FINE;
   1:  PR[GP1:91,1] = PR[GP1:90,1] + 93.680;
   1:  PR[GP1:91,2] = PR[GP1:90,2] + 121.972;
   1:L PR[91] 10mm/sec FINE;
   1:  PR[GP1:91,1] = PR[GP1:90,1] + 92.019;
   1:  PR[GP1:91,2] = PR[GP1:90,2] + 122.789;
   1:L PR[91] 10mm/sec FINE;
   1:  PR[GP1:91,1] = PR[GP1:90,1] + 89.569;
   1:  PR[GP1:91,2] = PR[GP1:90,2] + 123.795;
   1:L PR[91] 10mm/sec FINE;
   1:  PR[GP1:91,1] = PR[GP1:90,1] + 89.032;
   1:  PR[GP1:91,2] = PR[GP1:90,2] + 123.987;
   1:L PR[91] 10mm/sec FINE;
   1:  PR[GP1:91,1] = PR[GP1:90,1] + 87.873;
   1:  PR[GP1:91,2] = PR[GP1:90,2] + 124.268;
   1:L PR[91] 10mm/sec FINE;
   1:  PR[GP1:91,1] = PR[GP1:90,1] + 85.783;
   1:  PR[GP1:91,2] = PR[GP1:90,2] + 124.825;
   1:L PR[91] 10mm/sec FINE;
   1:  PR[GP1:91,1] = PR[GP1:90,1] + 84.622;
   1:  PR[GP1:91,2] = PR[GP1:90,2] + 125.031;
   1:L PR[91] 10mm/sec FINE;
   1:  PR[GP1:91,1] = PR[GP1:90,1] + 82.504;
   1:  PR[GP1:91,2] = PR[GP1:90,2] + 125.227;
   1:L PR[91] 10mm/sec FINE;
   1:  PR[GP1:91,1] = PR[GP1:90,1] + 79.761;
   1:  PR[GP1:91,2] = PR[GP1:90,2] + 125.217;
   1:L PR[91] 10mm/sec FINE;
   1:  PR[GP1:91,1] = PR[GP1:90,1] + 79.017;
   1:  PR[GP1:91,2] = PR[GP1:90,2] + 125.158;
   1:L PR[91] 10mm/sec FINE;
   1:  PR[GP1:91,1] = PR[GP1:90,1] + 76.700;
   1:  PR[GP1:91,2] = PR[GP1:90,2] + 124.718;
   1:L PR[91] 10mm/sec FINE;
   1:  PR[GP1:91,1] = PR[GP1:90,1] + 75.365;
   1:  PR[GP1:91,2] = PR[GP1:90,2] + 124.441;
   1:L PR[91] 10mm/sec FINE;
   1:  PR[GP1:91,1] = PR[GP1:90,1] + 72.691;
   1:  PR[GP1:91,2] = PR[GP1:90,2] + 123.312;
   1:L PR[91] 10mm/sec FINE;
   1:  PR[GP1:91,1] = PR[GP1:90,1] + 71.836;
   1:  PR[GP1:91,2] = PR[GP1:90,2] + 122.932;
   1:L PR[91] 10mm/sec FINE;
   1:  PR[GP1:91,1] = PR[GP1:90,1] + 69.949;
   1:  PR[GP1:91,2] = PR[GP1:90,2] + 121.623;
   1:L PR[91] 10mm/sec FINE;
   1:  PR[GP1:91,1] = PR[GP1:90,1] + 68.789;
   1:  PR[GP1:91,2] = PR[GP1:90,2] + 120.792;
   1:L PR[91] 10mm/sec FINE;
   1:  PR[GP1:91,1] = PR[GP1:90,1] + 66.339;
   1:  PR[GP1:91,2] = PR[GP1:90,2] + 118.114;
   1:L PR[91] 10mm/sec FINE;
   1:  PR[GP1:91,1] = PR[GP1:90,1] + 65.536;
   1:  PR[GP1:91,2] = PR[GP1:90,2] + 116.729;
   1:L PR[91] 10mm/sec FINE;
   1:  PR[GP1:91,1] = PR[GP1:90,1] + 64.556;
   1:  PR[GP1:91,2] = PR[GP1:90,2] + 115.019;
   1:L PR[91] 10mm/sec FINE;
   1:  PR[GP1:91,1] = PR[GP1:90,1] + 63.467;
   1:  PR[GP1:91,2] = PR[GP1:90,2] + 111.647;
   1:L PR[91] 10mm/sec FINE;
   1:  PR[GP1:91,1] = PR[GP1:90,1] + 63.220;
   1:  PR[GP1:91,2] = PR[GP1:90,2] + 108.076;
   1:L PR[91] 10mm/sec FINE;
   1:  PR[GP1:91,1] = PR[GP1:90,1] + 63.484;
   1:  PR[GP1:91,2] = PR[GP1:90,2] + 106.278;
   1:L PR[91] 10mm/sec FINE;
   1:  PR[GP1:91,1] = PR[GP1:90,1] + 63.779;
   1:  PR[GP1:91,2] = PR[GP1:90,2] + 104.434;
   1:L PR[91] 10mm/sec FINE;
   1:  PR[GP1:91,1] = PR[GP1:90,1] + 64.284;
   1:  PR[GP1:91,2] = PR[GP1:90,2] + 103.036;
   1:L PR[91] 10mm/sec FINE;
   1:  PR[GP1:91,1] = PR[GP1:90,1] + 65.072;
   1:  PR[GP1:91,2] = PR[GP1:90,2] + 100.935;
   1:L PR[91] 10mm/sec FINE;
   1:  PR[GP1:91,1] = PR[GP1:90,1] + 65.619;
   1:  PR[GP1:91,2] = PR[GP1:90,2] + 100.061;
   1:L PR[91] 10mm/sec FINE;
   1:  PR[GP1:91,1] = PR[GP1:90,1] + 67.191;
   1:  PR[GP1:91,2] = PR[GP1:90,2] + 97.669;
   1:L PR[91] 10mm/sec FINE;
   1:  PR[GP1:91,1] = PR[GP1:90,1] + 68.587;
   1:  PR[GP1:91,2] = PR[GP1:90,2] + 96.260;
   1:L PR[91] 10mm/sec FINE;
   1:  PR[GP1:91,1] = PR[GP1:90,1] + 70.028;
   1:  PR[GP1:91,2] = PR[GP1:90,2] + 94.877;
   1:L PR[91] 10mm/sec FINE;
   1:  PR[GP1:91,1] = PR[GP1:90,1] + 71.875;
   1:  PR[GP1:91,2] = PR[GP1:90,2] + 93.833;
   1:  PR[GP1:91,3] = PR[GP1:90,3] + 29.900;
   1:L PR[91] 10mm/sec FINE;
   1:  PR[GP1:91,1] = PR[GP1:90,1] + 73.694;
   1:  PR[GP1:91,2] = PR[GP1:90,2] + 92.649;
   1:L PR[91] 10mm/sec FINE;
   1:  PR[GP1:91,1] = PR[GP1:90,1] + 76.877;
   1:  PR[GP1:91,2] = PR[GP1:90,2] + 91.192;
   1:L PR[91] 10mm/sec FINE;
   1:  PR[GP1:91,1] = PR[GP1:90,1] + 77.071;
   1:  PR[GP1:91,2] = PR[GP1:90,2] + 91.111;
   1:L PR[91] 10mm/sec FINE;
   1:  PR[GP1:91,1] = PR[GP1:90,1] + 80.608;
   1:  PR[GP1:91,2] = PR[GP1:90,2] + 90.138;
   1:L PR[91] 10mm/sec FINE;
   1:  PR[GP1:91,1] = PR[GP1:90,1] + 82.092;
   1:  PR[GP1:91,2] = PR[GP1:90,2] + 89.865;
   1:L PR[91] 10mm/sec FINE;
   1:  PR[GP1:91,1] = PR[GP1:90,1] + 83.660;
   1:  PR[GP1:91,2] = PR[GP1:90,2] + 89.691;
   1:L PR[91] 10mm/sec FINE;
   1:  PR[GP1:91,1] = PR[GP1:90,1] + 85.917;
   1:  PR[GP1:91,2] = PR[GP1:90,2] + 89.567;
   1:L PR[91] 10mm/sec FINE;
   1:  PR[GP1:91,1] = PR[GP1:90,1] + 86.300;
   1:  PR[GP1:91,2] = PR[GP1:90,2] + 89.533;
   1:L PR[91] 10mm/sec FINE;
   1:  PR[GP1:91,1] = PR[GP1:90,1] + 86.411;
   1:  PR[GP1:91,2] = PR[GP1:90,2] + 89.528;
   1:L PR[91] 10mm/sec FINE;
   1:  PR[GP1:91,1] = PR[GP1:90,1] + 89.621;
   1:  PR[GP1:91,2] = PR[GP1:90,2] + 89.644;
   1:L PR[91] 10mm/sec FINE;
   1:  PR[GP1:91,1] = PR[GP1:90,1] + 90.813;
   1:  PR[GP1:91,2] = PR[GP1:90,2] + 89.815;
   1:L PR[91] 10mm/sec FINE;
   1:  PR[GP1:91,1] = PR[GP1:90,1] + 93.394;
   1:  PR[GP1:91,2] = PR[GP1:90,2] + 90.271;
   1:L PR[91] 10mm/sec FINE;
   1:  PR[GP1:91,1] = PR[GP1:90,1] + 95.230;
   1:  PR[GP1:91,2] = PR[GP1:90,2] + 90.883;
   1:L PR[91] 10mm/sec FINE;
   1:  PR[GP1:91,1] = PR[GP1:90,1] + 96.110;
   1:  PR[GP1:91,2] = PR[GP1:90,2] + 91.242;
   1:L PR[91] 10mm/sec FINE;
   1:  PR[GP1:91,1] = PR[GP1:90,1] + 96.654;
   1:  PR[GP1:91,2] = PR[GP1:90,2] + 91.371;
   1:L PR[91] 10mm/sec FINE;
   1:  PR[GP1:91,1] = PR[GP1:90,1] + 97.860;
   1:  PR[GP1:91,2] = PR[GP1:90,2] + 91.119;
   1:L PR[91] 10mm/sec FINE;
   1:  PR[GP1:91,1] = PR[GP1:90,1] + 98.968;
   1:  PR[GP1:91,2] = PR[GP1:90,2] + 90.607;
   1:L PR[91] 10mm/sec FINE;
   1:  PR[GP1:91,1] = PR[GP1:90,1] + 100.300;
   1:  PR[GP1:91,2] = PR[GP1:90,2] + 90.160;
   1:L PR[91] 10mm/sec FINE;
   1:  PR[GP1:91,1] = PR[GP1:90,1] + 101.657;
   1:  PR[GP1:91,2] = PR[GP1:90,2] + 89.684;
   1:L PR[91] 10mm/sec FINE;
   1:  PR[GP1:91,1] = PR[GP1:90,1] + 104.486;
   1:  PR[GP1:91,2] = PR[GP1:90,2] + 89.206;
   1:L PR[91] 10mm/sec FINE;
   1:  PR[GP1:91,1] = PR[GP1:90,1] + 107.389;
   1:  PR[GP1:91,2] = PR[GP1:90,2] + 89.194;
   1:L PR[91] 10mm/sec FINE;
   1:  PR[GP1:91,1] = PR[GP1:90,1] + 110.290;
   1:  PR[GP1:91,2] = PR[GP1:90,2] + 89.653;
   1:L PR[91] 10mm/sec FINE;
   1:  PR[GP1:91,1] = PR[GP1:90,1] + 111.064;
   1:  PR[GP1:91,2] = PR[GP1:90,2] + 89.906;
   1:L PR[91] 10mm/sec FINE;
   1:  PR[GP1:91,1] = PR[GP1:90,1] + 112.926;
   1:  PR[GP1:91,2] = PR[GP1:90,2] + 90.470;
   1:L PR[91] 10mm/sec FINE;
   1:  PR[GP1:91,1] = PR[GP1:90,1] + 113.392;
   1:  PR[GP1:91,2] = PR[GP1:90,2] + 90.655;
   1:L PR[91] 10mm/sec FINE;
   1:  PR[GP1:91,1] = PR[GP1:90,1] + 115.267;
   1:  PR[GP1:91,2] = PR[GP1:90,2] + 91.546;
   1:L PR[91] 10mm/sec FINE;
   1:  PR[GP1:91,1] = PR[GP1:90,1] + 116.377;
   1:  PR[GP1:91,2] = PR[GP1:90,2] + 92.180;
   1:L PR[91] 10mm/sec FINE;
   1:  PR[GP1:91,1] = PR[GP1:90,1] + 117.363;
   1:  PR[GP1:91,2] = PR[GP1:90,2] + 92.844;
   1:L PR[91] 10mm/sec FINE;
   1:  PR[GP1:91,1] = PR[GP1:90,1] + 119.008;
   1:  PR[GP1:91,2] = PR[GP1:90,2] + 94.122;
   1:L PR[91] 10mm/sec FINE;
   1:  PR[GP1:91,1] = PR[GP1:90,1] + 119.214;
   1:  PR[GP1:91,2] = PR[GP1:90,2] + 94.311;
   1:L PR[91] 10mm/sec FINE;
   1:  PR[GP1:91,1] = PR[GP1:90,1] + 119.757;
   1:  PR[GP1:91,2] = PR[GP1:90,2] + 94.871;
   1:L PR[91] 10mm/sec FINE;
   1:  PR[GP1:91,1] = PR[GP1:90,1] + 121.091;
   1:  PR[GP1:91,2] = PR[GP1:90,2] + 96.160;
   1:L PR[91] 10mm/sec FINE;
   1:  PR[GP1:91,1] = PR[GP1:90,1] + 122.793;
   1:  PR[GP1:91,2] = PR[GP1:90,2] + 98.347;
   1:L PR[91] 10mm/sec FINE;
   1:  PR[GP1:91,1] = PR[GP1:90,1] + 124.164;
   1:  PR[GP1:91,2] = PR[GP1:90,2] + 100.750;
   1:L PR[91] 10mm/sec FINE;
   1:  PR[GP1:91,1] = PR[GP1:90,1] + 125.168;
   1:  PR[GP1:91,2] = PR[GP1:90,2] + 103.314;
   1:L PR[91] 10mm/sec FINE;
   1:  PR[GP1:91,1] = PR[GP1:90,1] + 125.783;
   1:  PR[GP1:91,2] = PR[GP1:90,2] + 105.969;
   1:L PR[91] 10mm/sec FINE;
   1:  PR[GP1:91,1] = PR[GP1:90,1] + 125.960;
   1:  PR[GP1:91,2] = PR[GP1:90,2] + 108.666;
   1:L PR[91] 10mm/sec FINE;
   1:  PR[GP1:91,1] = PR[GP1:90,1] + 125.551;
   1:  PR[GP1:91,2] = PR[GP1:90,2] + 112.143;
   1:L PR[91] 10mm/sec FINE;
   1:  PR[GP1:91,1] = PR[GP1:90,1] + 124.426;
   1:  PR[GP1:91,2] = PR[GP1:90,2] + 115.437;
   1:L PR[91] 10mm/sec FINE;
   1:  PR[GP1:91,1] = PR[GP1:90,1] + 122.624;
   1:  PR[GP1:91,2] = PR[GP1:90,2] + 118.419;
   1:L PR[91] 10mm/sec FINE;
   1:  PR[GP1:91,1] = PR[GP1:90,1] + 120.221;
   1:  PR[GP1:91,2] = PR[GP1:90,2] + 120.984;
   1:L PR[91] 10mm/sec FINE;
   1:  PR[GP1:91,1] = PR[GP1:90,1] + 117.314;
   1:  PR[GP1:91,2] = PR[GP1:90,2] + 123.036;
   1:L PR[91] 10mm/sec FINE;
   1:  PR[GP1:91,1] = PR[GP1:90,1] + 114.021;
   1:  PR[GP1:91,2] = PR[GP1:90,2] + 124.501;
   1:L PR[91] 10mm/sec FINE;
   1:  PR[GP1:91,1] = PR[GP1:90,1] + 110.528;
   1:  PR[GP1:91,2] = PR[GP1:90,2] + 125.304;
   1:L PR[91] 10mm/sec FINE;
   1:  PR[GP1:91,1] = PR[GP1:90,1] + 108.849;
   1:  PR[GP1:91,2] = PR[GP1:90,2] + 125.374;
   1:L PR[91] 10mm/sec FINE;
   1:  PR[GP1:91,1] = PR[GP1:90,1] + 106.911;
   1:  PR[GP1:91,2] = PR[GP1:90,2] + 125.446;
   1:L PR[91] 10mm/sec FINE;
   1:  PR[GP1:91,1] = PR[GP1:90,1] + 103.291;
   1:  PR[GP1:91,2] = PR[GP1:90,2] + 124.929;
   1:L PR[91] 10mm/sec FINE;
   1:  PR[GP1:91,1] = PR[GP1:90,1] + 99.885;
   1:  PR[GP1:91,2] = PR[GP1:90,2] + 123.747;
   1:L PR[91] 10mm/sec FINE;
   1:  PR[GP1:91,1] = PR[GP1:90,1] + 98.993;
   1:  PR[GP1:91,2] = PR[GP1:90,2] + 123.283;
   1:L PR[91] 10mm/sec FINE;
   1:  PR[GP1:91,1] = PR[GP1:90,1] + 96.672;
   1:  PR[GP1:91,2] = PR[GP1:90,2] + 121.976;
   1:L PR[91] 10mm/sec FINE;
   1:  PR[GP1:91,1] = PR[GP1:90,1] + 95.683;
   1:  PR[GP1:91,2] = PR[GP1:90,2] + 121.594;
   1:L PR[91] 10mm/sec FINE;
   1:  PR[GP1:91,1] = PR[GP1:90,1] + 95.523;
   1:  PR[GP1:91,2] = PR[GP1:90,2] + 121.578;
   1:L PR[91] 10mm/sec FINE;
   1:  PR[GP1:91,1] = PR[GP1:90,1] + 95.225;
   1:  PR[GP1:91,2] = PR[GP1:90,2] + 121.644;
   1:L PR[91] 10mm/sec FINE;
   1:  PR[GP1:91,1] = PR[GP1:90,1] + 94.608;
   1:  PR[GP1:91,2] = PR[GP1:90,2] + 121.731;
   1:L PR[91] 10mm/sec FINE;
   1:  PR[GP1:91,1] = PR[GP1:90,1] + 93.951;
   1:  PR[GP1:91,2] = PR[GP1:90,2] + 122.026;
   1:L PR[91] 10mm/sec FINE;
   1:  PR[GP1:91,1] = PR[GP1:90,1] + 92.336;
   1:  PR[GP1:91,2] = PR[GP1:90,2] + 122.820;
   1:L PR[91] 10mm/sec FINE;
   1:  PR[GP1:91,1] = PR[GP1:90,1] + 91.000;
   1:  PR[GP1:91,2] = PR[GP1:90,2] + 123.368;
   1:L PR[91] 10mm/sec FINE;
   1:  PR[GP1:91,1] = PR[GP1:90,1] + 89.547;
   1:  PR[GP1:91,2] = PR[GP1:90,2] + 123.889;
   1:L PR[91] 10mm/sec FINE;
   1:  PR[GP1:91,1] = PR[GP1:90,1] + 86.452;
   1:  PR[GP1:91,2] = PR[GP1:90,2] + 124.639;
   1:L PR[91] 10mm/sec FINE;
   1:  PR[GP1:91,1] = PR[GP1:90,1] + 85.934;
   1:  PR[GP1:91,2] = PR[GP1:90,2] + 124.777;
   1:L PR[91] 10mm/sec FINE;
   1:  PR[GP1:91,1] = PR[GP1:90,1] + 85.656;
   1:  PR[GP1:91,2] = PR[GP1:90,2] + 124.826;
   1:L PR[91] 10mm/sec FINE;
   1:  PR[GP1:91,1] = PR[GP1:90,1] + 82.705;
   1:  PR[GP1:91,2] = PR[GP1:90,2] + 125.100;
   1:L PR[91] 10mm/sec FINE;
   1:  PR[GP1:91,1] = PR[GP1:90,1] + 80.816;
   1:  PR[GP1:91,2] = PR[GP1:90,2] + 125.093;
   1:L PR[91] 10mm/sec FINE;
   1:  PR[GP1:91,1] = PR[GP1:90,1] + 79.275;
   1:  PR[GP1:91,2] = PR[GP1:90,2] + 124.971;
   1:L PR[91] 10mm/sec FINE;
   1:  PR[GP1:91,1] = PR[GP1:90,1] + 76.114;
   1:  PR[GP1:91,2] = PR[GP1:90,2] + 124.370;
   1:L PR[91] 10mm/sec FINE;
   1:  PR[GP1:91,1] = PR[GP1:90,1] + 75.774;
   1:  PR[GP1:91,2] = PR[GP1:90,2] + 124.280;
   1:L PR[91] 10mm/sec FINE;
   1:  PR[GP1:91,1] = PR[GP1:90,1] + 74.472;
   1:  PR[GP1:91,2] = PR[GP1:90,2] + 123.760;
   1:L PR[91] 10mm/sec FINE;
   1:  PR[GP1:91,1] = PR[GP1:90,1] + 72.302;
   1:  PR[GP1:91,2] = PR[GP1:90,2] + 122.835;
   1:L PR[91] 10mm/sec FINE;
   1:  PR[GP1:91,1] = PR[GP1:90,1] + 69.976;
   1:  PR[GP1:91,2] = PR[GP1:90,2] + 121.221;
   1:L PR[91] 10mm/sec FINE;
   1:  PR[GP1:91,1] = PR[GP1:90,1] + 69.239;
   1:  PR[GP1:91,2] = PR[GP1:90,2] + 120.693;
   1:L PR[91] 10mm/sec FINE;
   1:  PR[GP1:91,1] = PR[GP1:90,1] + 66.776;
   1:  PR[GP1:91,2] = PR[GP1:90,2] + 118.008;
   1:L PR[91] 10mm/sec FINE;
   1:  PR[GP1:91,1] = PR[GP1:90,1] + 64.984;
   1:  PR[GP1:91,2] = PR[GP1:90,2] + 114.903;
   1:L PR[91] 10mm/sec FINE;
   1:  PR[GP1:91,1] = PR[GP1:90,1] + 63.889;
   1:  PR[GP1:91,2] = PR[GP1:90,2] + 111.520;
   1:L PR[91] 10mm/sec FINE;
   1:  PR[GP1:91,1] = PR[GP1:90,1] + 63.644;
   1:  PR[GP1:91,2] = PR[GP1:90,2] + 107.936;
   1:L PR[91] 10mm/sec FINE;
   1:  PR[GP1:91,1] = PR[GP1:90,1] + 63.834;
   1:  PR[GP1:91,2] = PR[GP1:90,2] + 106.646;
   1:L PR[91] 10mm/sec FINE;
   1:  PR[GP1:91,1] = PR[GP1:90,1] + 64.212;
   1:  PR[GP1:91,2] = PR[GP1:90,2] + 104.277;
   1:L PR[91] 10mm/sec FINE;
   1:  PR[GP1:91,1] = PR[GP1:90,1] + 65.518;
   1:  PR[GP1:91,2] = PR[GP1:90,2] + 100.762;
   1:L PR[91] 10mm/sec FINE;
   1:  PR[GP1:91,1] = PR[GP1:90,1] + 65.782;
   1:  PR[GP1:91,2] = PR[GP1:90,2] + 100.341;
   1:L PR[91] 10mm/sec FINE;
   1:  PR[GP1:91,1] = PR[GP1:90,1] + 67.186;
   1:  PR[GP1:91,2] = PR[GP1:90,2] + 98.203;
   1:L PR[91] 10mm/sec FINE;
   1:  PR[GP1:91,1] = PR[GP1:90,1] + 67.667;
   1:  PR[GP1:91,2] = PR[GP1:90,2] + 97.510;
   1:L PR[91] 10mm/sec FINE;
   1:  PR[GP1:91,1] = PR[GP1:90,1] + 70.498;
   1:  PR[GP1:91,2] = PR[GP1:90,2] + 94.787;
   1:L PR[91] 10mm/sec FINE;
   1:  PR[GP1:91,1] = PR[GP1:90,1] + 73.143;
   1:  PR[GP1:91,2] = PR[GP1:90,2] + 93.191;
   1:  PR[GP1:91,3] = PR[GP1:90,3] + 30.900;
   1:L PR[91] 10mm/sec FINE;
   1:  PR[GP1:91,1] = PR[GP1:90,1] + 74.109;
   1:  PR[GP1:91,2] = PR[GP1:90,2] + 92.561;
   1:L PR[91] 10mm/sec FINE;
   1:  PR[GP1:91,1] = PR[GP1:90,1] + 77.578;
   1:  PR[GP1:91,2] = PR[GP1:90,2] + 90.980;
   1:L PR[91] 10mm/sec FINE;
   1:  PR[GP1:91,1] = PR[GP1:90,1] + 78.308;
   1:  PR[GP1:91,2] = PR[GP1:90,2] + 90.746;
   1:L PR[91] 10mm/sec FINE;
   1:  PR[GP1:91,1] = PR[GP1:90,1] + 80.981;
   1:  PR[GP1:91,2] = PR[GP1:90,2] + 90.006;
   1:L PR[91] 10mm/sec FINE;
   1:  PR[GP1:91,1] = PR[GP1:90,1] + 83.308;
   1:  PR[GP1:91,2] = PR[GP1:90,2] + 89.579;
   1:L PR[91] 10mm/sec FINE;
   1:  PR[GP1:91,1] = PR[GP1:90,1] + 83.875;
   1:  PR[GP1:91,2] = PR[GP1:90,2] + 89.516;
   1:L PR[91] 10mm/sec FINE;
   1:  PR[GP1:91,1] = PR[GP1:90,1] + 84.701;
   1:  PR[GP1:91,2] = PR[GP1:90,2] + 89.471;
   1:L PR[91] 10mm/sec FINE;
   1:  PR[GP1:91,1] = PR[GP1:90,1] + 86.803;
   1:  PR[GP1:91,2] = PR[GP1:90,2] + 89.286;
   1:L PR[91] 10mm/sec FINE;
   1:  PR[GP1:91,1] = PR[GP1:90,1] + 87.467;
   1:  PR[GP1:91,2] = PR[GP1:90,2] + 89.251;
   1:L PR[91] 10mm/sec FINE;
   1:  PR[GP1:91,1] = PR[GP1:90,1] + 90.284;
   1:  PR[GP1:91,2] = PR[GP1:90,2] + 89.353;
   1:L PR[91] 10mm/sec FINE;
   1:  PR[GP1:91,1] = PR[GP1:90,1] + 92.100;
   1:  PR[GP1:91,2] = PR[GP1:90,2] + 89.613;
   1:L PR[91] 10mm/sec FINE;
   1:  PR[GP1:91,1] = PR[GP1:90,1] + 94.236;
   1:  PR[GP1:91,2] = PR[GP1:90,2] + 89.990;
   1:L PR[91] 10mm/sec FINE;
   1:  PR[GP1:91,1] = PR[GP1:90,1] + 95.800;
   1:  PR[GP1:91,2] = PR[GP1:90,2] + 90.513;
   1:L PR[91] 10mm/sec FINE;
   1:  PR[GP1:91,1] = PR[GP1:90,1] + 96.454;
   1:  PR[GP1:91,2] = PR[GP1:90,2] + 90.770;
   1:L PR[91] 10mm/sec FINE;
   1:  PR[GP1:91,1] = PR[GP1:90,1] + 96.905;
   1:  PR[GP1:91,2] = PR[GP1:90,2] + 90.878;
   1:L PR[91] 10mm/sec FINE;
   1:  PR[GP1:91,1] = PR[GP1:90,1] + 98.114;
   1:  PR[GP1:91,2] = PR[GP1:90,2] + 90.656;
   1:L PR[91] 10mm/sec FINE;
   1:  PR[GP1:91,1] = PR[GP1:90,1] + 98.726;
   1:  PR[GP1:91,2] = PR[GP1:90,2] + 90.384;
   1:L PR[91] 10mm/sec FINE;
   1:  PR[GP1:91,1] = PR[GP1:90,1] + 101.409;
   1:  PR[GP1:91,2] = PR[GP1:90,2] + 89.453;
   1:L PR[91] 10mm/sec FINE;
   1:  PR[GP1:91,1] = PR[GP1:90,1] + 104.235;
   1:  PR[GP1:91,2] = PR[GP1:90,2] + 88.966;
   1:L PR[91] 10mm/sec FINE;
   1:  PR[GP1:91,1] = PR[GP1:90,1] + 107.135;
   1:  PR[GP1:91,2] = PR[GP1:90,2] + 88.942;
   1:L PR[91] 10mm/sec FINE;
   1:  PR[GP1:91,1] = PR[GP1:90,1] + 110.035;
   1:  PR[GP1:91,2] = PR[GP1:90,2] + 89.388;
   1:L PR[91] 10mm/sec FINE;
   1:  PR[GP1:91,1] = PR[GP1:90,1] + 112.858;
   1:  PR[GP1:91,2] = PR[GP1:90,2] + 90.303;
   1:L PR[91] 10mm/sec FINE;
   1:  PR[GP1:91,1] = PR[GP1:90,1] + 114.110;
   1:  PR[GP1:91,2] = PR[GP1:90,2] + 90.939;
   1:L PR[91] 10mm/sec FINE;
   1:  PR[GP1:91,1] = PR[GP1:90,1] + 115.374;
   1:  PR[GP1:91,2] = PR[GP1:90,2] + 91.540;
   1:L PR[91] 10mm/sec FINE;
   1:  PR[GP1:91,1] = PR[GP1:90,1] + 115.715;
   1:  PR[GP1:91,2] = PR[GP1:90,2] + 91.735;
   1:L PR[91] 10mm/sec FINE;
   1:  PR[GP1:91,1] = PR[GP1:90,1] + 117.486;
   1:  PR[GP1:91,2] = PR[GP1:90,2] + 92.928;
   1:L PR[91] 10mm/sec FINE;
   1:  PR[GP1:91,1] = PR[GP1:90,1] + 118.424;
   1:  PR[GP1:91,2] = PR[GP1:90,2] + 93.656;
   1:L PR[91] 10mm/sec FINE;
   1:  PR[GP1:91,1] = PR[GP1:90,1] + 119.333;
   1:  PR[GP1:91,2] = PR[GP1:90,2] + 94.490;
   1:L PR[91] 10mm/sec FINE;
   1:  PR[GP1:91,1] = PR[GP1:90,1] + 120.705;
   1:  PR[GP1:91,2] = PR[GP1:90,2] + 95.907;
   1:L PR[91] 10mm/sec FINE;
   1:  PR[GP1:91,1] = PR[GP1:90,1] + 120.926;
   1:  PR[GP1:91,2] = PR[GP1:90,2] + 96.182;
   1:L PR[91] 10mm/sec FINE;
   1:  PR[GP1:91,1] = PR[GP1:90,1] + 121.536;
   1:  PR[GP1:91,2] = PR[GP1:90,2] + 97.023;
   1:L PR[91] 10mm/sec FINE;
   1:  PR[GP1:91,1] = PR[GP1:90,1] + 122.468;
   1:  PR[GP1:91,2] = PR[GP1:90,2] + 98.226;
   1:L PR[91] 10mm/sec FINE;
   1:  PR[GP1:91,1] = PR[GP1:90,1] + 123.826;
   1:  PR[GP1:91,2] = PR[GP1:90,2] + 100.620;
   1:L PR[91] 10mm/sec FINE;
   1:  PR[GP1:91,1] = PR[GP1:90,1] + 124.326;
   1:  PR[GP1:91,2] = PR[GP1:90,2] + 101.897;
   1:L PR[91] 10mm/sec FINE;
   1:  PR[GP1:91,1] = PR[GP1:90,1] + 124.821;
   1:  PR[GP1:91,2] = PR[GP1:90,2] + 103.174;
   1:L PR[91] 10mm/sec FINE;
   1:  PR[GP1:91,1] = PR[GP1:90,1] + 125.418;
   1:  PR[GP1:91,2] = PR[GP1:90,2] + 105.828;
   1:L PR[91] 10mm/sec FINE;
   1:  PR[GP1:91,1] = PR[GP1:90,1] + 125.568;
   1:  PR[GP1:91,2] = PR[GP1:90,2] + 108.532;
   1:L PR[91] 10mm/sec FINE;
   1:  PR[GP1:91,1] = PR[GP1:90,1] + 125.167;
   1:  PR[GP1:91,2] = PR[GP1:90,2] + 112.010;
   1:L PR[91] 10mm/sec FINE;
   1:  PR[GP1:91,1] = PR[GP1:90,1] + 124.043;
   1:  PR[GP1:91,2] = PR[GP1:90,2] + 115.307;
   1:L PR[91] 10mm/sec FINE;
   1:  PR[GP1:91,1] = PR[GP1:90,1] + 122.238;
   1:  PR[GP1:91,2] = PR[GP1:90,2] + 118.295;
   1:L PR[91] 10mm/sec FINE;
   1:  PR[GP1:91,1] = PR[GP1:90,1] + 119.831;
   1:  PR[GP1:91,2] = PR[GP1:90,2] + 120.863;
   1:L PR[91] 10mm/sec FINE;
   1:  PR[GP1:91,1] = PR[GP1:90,1] + 116.918;
   1:  PR[GP1:91,2] = PR[GP1:90,2] + 122.920;
   1:L PR[91] 10mm/sec FINE;
   1:  PR[GP1:91,1] = PR[GP1:90,1] + 113.689;
   1:  PR[GP1:91,2] = PR[GP1:90,2] + 124.358;
   1:L PR[91] 10mm/sec FINE;
   1:  PR[GP1:91,1] = PR[GP1:90,1] + 110.177;
   1:  PR[GP1:91,2] = PR[GP1:90,2] + 125.171;
   1:L PR[91] 10mm/sec FINE;
   1:  PR[GP1:91,1] = PR[GP1:90,1] + 106.582;
   1:  PR[GP1:91,2] = PR[GP1:90,2] + 125.309;
   1:L PR[91] 10mm/sec FINE;
   1:  PR[GP1:91,1] = PR[GP1:90,1] + 104.961;
   1:  PR[GP1:91,2] = PR[GP1:90,2] + 125.082;
   1:L PR[91] 10mm/sec FINE;
   1:  PR[GP1:91,1] = PR[GP1:90,1] + 103.020;
   1:  PR[GP1:91,2] = PR[GP1:90,2] + 124.780;
   1:L PR[91] 10mm/sec FINE;
   1:  PR[GP1:91,1] = PR[GP1:90,1] + 99.612;
   1:  PR[GP1:91,2] = PR[GP1:90,2] + 123.602;
   1:L PR[91] 10mm/sec FINE;
   1:  PR[GP1:91,1] = PR[GP1:90,1] + 98.151;
   1:  PR[GP1:91,2] = PR[GP1:90,2] + 122.842;
   1:L PR[91] 10mm/sec FINE;
   1:  PR[GP1:91,1] = PR[GP1:90,1] + 96.808;
   1:  PR[GP1:91,2] = PR[GP1:90,2] + 122.087;
   1:L PR[91] 10mm/sec FINE;
   1:  PR[GP1:91,1] = PR[GP1:90,1] + 96.173;
   1:  PR[GP1:91,2] = PR[GP1:90,2] + 121.901;
   1:L PR[91] 10mm/sec FINE;
   1:  PR[GP1:91,1] = PR[GP1:90,1] + 95.756;
   1:  PR[GP1:91,2] = PR[GP1:90,2] + 121.740;
   1:L PR[91] 10mm/sec FINE;
   1:  PR[GP1:91,1] = PR[GP1:90,1] + 95.656;
   1:  PR[GP1:91,2] = PR[GP1:90,2] + 121.730;
   1:L PR[91] 10mm/sec FINE;
   1:  PR[GP1:91,1] = PR[GP1:90,1] + 94.663;
   1:  PR[GP1:91,2] = PR[GP1:90,2] + 121.942;
   1:L PR[91] 10mm/sec FINE;
   1:  PR[GP1:91,1] = PR[GP1:90,1] + 92.428;
   1:  PR[GP1:91,2] = PR[GP1:90,2] + 122.943;
   1:L PR[91] 10mm/sec FINE;
   1:  PR[GP1:91,1] = PR[GP1:90,1] + 90.062;
   1:  PR[GP1:91,2] = PR[GP1:90,2] + 123.790;
   1:L PR[91] 10mm/sec FINE;
   1:  PR[GP1:91,1] = PR[GP1:90,1] + 86.511;
   1:  PR[GP1:91,2] = PR[GP1:90,2] + 124.641;
   1:L PR[91] 10mm/sec FINE;
   1:  PR[GP1:91,1] = PR[GP1:90,1] + 82.906;
   1:  PR[GP1:91,2] = PR[GP1:90,2] + 124.972;
   1:L PR[91] 10mm/sec FINE;
   1:  PR[GP1:91,1] = PR[GP1:90,1] + 81.871;
   1:  PR[GP1:91,2] = PR[GP1:90,2] + 124.968;
   1:L PR[91] 10mm/sec FINE;
   1:  PR[GP1:91,1] = PR[GP1:90,1] + 79.534;
   1:  PR[GP1:91,2] = PR[GP1:90,2] + 124.783;
   1:L PR[91] 10mm/sec FINE;
   1:  PR[GP1:91,1] = PR[GP1:90,1] + 77.164;
   1:  PR[GP1:91,2] = PR[GP1:90,2] + 124.333;
   1:L PR[91] 10mm/sec FINE;
   1:  PR[GP1:91,1] = PR[GP1:90,1] + 76.095;
   1:  PR[GP1:91,2] = PR[GP1:90,2] + 124.051;
   1:L PR[91] 10mm/sec FINE;
   1:  PR[GP1:91,1] = PR[GP1:90,1] + 72.747;
   1:  PR[GP1:91,2] = PR[GP1:90,2] + 122.702;
   1:L PR[91] 10mm/sec FINE;
   1:  PR[GP1:91,1] = PR[GP1:90,1] + 72.087;
   1:  PR[GP1:91,2] = PR[GP1:90,2] + 122.266;
   1:L PR[91] 10mm/sec FINE;
   1:  PR[GP1:91,1] = PR[GP1:90,1] + 69.687;
   1:  PR[GP1:91,2] = PR[GP1:90,2] + 120.593;
   1:L PR[91] 10mm/sec FINE;
   1:  PR[GP1:91,1] = PR[GP1:90,1] + 67.213;
   1:  PR[GP1:91,2] = PR[GP1:90,2] + 117.902;
   1:L PR[91] 10mm/sec FINE;
   1:  PR[GP1:91,1] = PR[GP1:90,1] + 65.412;
   1:  PR[GP1:91,2] = PR[GP1:90,2] + 114.787;
   1:L PR[91] 10mm/sec FINE;
   1:  PR[GP1:91,1] = PR[GP1:90,1] + 64.311;
   1:  PR[GP1:91,2] = PR[GP1:90,2] + 111.393;
   1:L PR[91] 10mm/sec FINE;
   1:  PR[GP1:91,1] = PR[GP1:90,1] + 64.068;
   1:  PR[GP1:91,2] = PR[GP1:90,2] + 107.796;
   1:L PR[91] 10mm/sec FINE;
   1:  PR[GP1:91,1] = PR[GP1:90,1] + 64.645;
   1:  PR[GP1:91,2] = PR[GP1:90,2] + 104.118;
   1:L PR[91] 10mm/sec FINE;
   1:  PR[GP1:91,1] = PR[GP1:90,1] + 64.800;
   1:  PR[GP1:91,2] = PR[GP1:90,2] + 103.689;
   1:L PR[91] 10mm/sec FINE;
   1:  PR[GP1:91,1] = PR[GP1:90,1] + 65.933;
   1:  PR[GP1:91,2] = PR[GP1:90,2] + 100.670;
   1:L PR[91] 10mm/sec FINE;
   1:  PR[GP1:91,1] = PR[GP1:90,1] + 65.962;
   1:  PR[GP1:91,2] = PR[GP1:90,2] + 100.598;
   1:L PR[91] 10mm/sec FINE;
   1:  PR[GP1:91,1] = PR[GP1:90,1] + 68.181;
   1:  PR[GP1:91,2] = PR[GP1:90,2] + 97.405;
   1:L PR[91] 10mm/sec FINE;
   1:  PR[GP1:91,1] = PR[GP1:90,1] + 68.971;
   1:  PR[GP1:91,2] = PR[GP1:90,2] + 96.613;
   1:L PR[91] 10mm/sec FINE;
   1:  PR[GP1:91,1] = PR[GP1:90,1] + 70.967;
   1:  PR[GP1:91,2] = PR[GP1:90,2] + 94.697;
   1:L PR[91] 10mm/sec FINE;
   1:  PR[GP1:91,1] = PR[GP1:90,1] + 74.410;
   1:  PR[GP1:91,2] = PR[GP1:90,2] + 92.549;
   1:  PR[GP1:91,3] = PR[GP1:90,3] + 31.900;
   1:L PR[91] 10mm/sec FINE;
   1:  PR[GP1:91,1] = PR[GP1:90,1] + 74.525;
   1:  PR[GP1:91,2] = PR[GP1:90,2] + 92.474;
   1:L PR[91] 10mm/sec FINE;
   1:  PR[GP1:91,1] = PR[GP1:90,1] + 78.115;
   1:  PR[GP1:91,2] = PR[GP1:90,2] + 90.844;
   1:L PR[91] 10mm/sec FINE;
   1:  PR[GP1:91,1] = PR[GP1:90,1] + 79.784;
   1:  PR[GP1:91,2] = PR[GP1:90,2] + 90.309;
   1:L PR[91] 10mm/sec FINE;
   1:  PR[GP1:91,1] = PR[GP1:90,1] + 81.353;
   1:  PR[GP1:91,2] = PR[GP1:90,2] + 89.875;
   1:L PR[91] 10mm/sec FINE;
   1:  PR[GP1:91,1] = PR[GP1:90,1] + 83.536;
   1:  PR[GP1:91,2] = PR[GP1:90,2] + 89.475;
   1:L PR[91] 10mm/sec FINE;
   1:  PR[GP1:91,1] = PR[GP1:90,1] + 84.364;
   1:  PR[GP1:91,2] = PR[GP1:90,2] + 89.297;
   1:L PR[91] 10mm/sec FINE;
   1:  PR[GP1:91,1] = PR[GP1:90,1] + 87.306;
   1:  PR[GP1:91,2] = PR[GP1:90,2] + 89.038;
   1:L PR[91] 10mm/sec FINE;
   1:  PR[GP1:91,1] = PR[GP1:90,1] + 88.523;
   1:  PR[GP1:91,2] = PR[GP1:90,2] + 88.974;
   1:L PR[91] 10mm/sec FINE;
   1:  PR[GP1:91,1] = PR[GP1:90,1] + 90.947;
   1:  PR[GP1:91,2] = PR[GP1:90,2] + 89.062;
   1:L PR[91] 10mm/sec FINE;
   1:  PR[GP1:91,1] = PR[GP1:90,1] + 93.388;
   1:  PR[GP1:91,2] = PR[GP1:90,2] + 89.411;
   1:L PR[91] 10mm/sec FINE;
   1:  PR[GP1:91,1] = PR[GP1:90,1] + 95.079;
   1:  PR[GP1:91,2] = PR[GP1:90,2] + 89.710;
   1:L PR[91] 10mm/sec FINE;
   1:  PR[GP1:91,1] = PR[GP1:90,1] + 96.370;
   1:  PR[GP1:91,2] = PR[GP1:90,2] + 90.142;
   1:L PR[91] 10mm/sec FINE;
   1:  PR[GP1:91,1] = PR[GP1:90,1] + 96.809;
   1:  PR[GP1:91,2] = PR[GP1:90,2] + 90.309;
   1:L PR[91] 10mm/sec FINE;
   1:  PR[GP1:91,1] = PR[GP1:90,1] + 97.167;
   1:  PR[GP1:91,2] = PR[GP1:90,2] + 90.393;
   1:L PR[91] 10mm/sec FINE;
   1:  PR[GP1:91,1] = PR[GP1:90,1] + 98.376;
   1:  PR[GP1:91,2] = PR[GP1:90,2] + 90.207;
   1:L PR[91] 10mm/sec FINE;
   1:  PR[GP1:91,1] = PR[GP1:90,1] + 101.162;
   1:  PR[GP1:91,2] = PR[GP1:90,2] + 89.223;
   1:L PR[91] 10mm/sec FINE;
   1:  PR[GP1:91,1] = PR[GP1:90,1] + 103.984;
   1:  PR[GP1:91,2] = PR[GP1:90,2] + 88.725;
   1:L PR[91] 10mm/sec FINE;
   1:  PR[GP1:91,1] = PR[GP1:90,1] + 106.882;
   1:  PR[GP1:91,2] = PR[GP1:90,2] + 88.690;
   1:L PR[91] 10mm/sec FINE;
   1:  PR[GP1:91,1] = PR[GP1:90,1] + 109.780;
   1:  PR[GP1:91,2] = PR[GP1:90,2] + 89.123;
   1:L PR[91] 10mm/sec FINE;
   1:  PR[GP1:91,1] = PR[GP1:90,1] + 112.604;
   1:  PR[GP1:91,2] = PR[GP1:90,2] + 90.024;
   1:L PR[91] 10mm/sec FINE;
   1:  PR[GP1:91,1] = PR[GP1:90,1] + 115.277;
   1:  PR[GP1:91,2] = PR[GP1:90,2] + 91.372;
   1:L PR[91] 10mm/sec FINE;
   1:  PR[GP1:91,1] = PR[GP1:90,1] + 116.778;
   1:  PR[GP1:91,2] = PR[GP1:90,2] + 92.452;
   1:L PR[91] 10mm/sec FINE;
   1:  PR[GP1:91,1] = PR[GP1:90,1] + 117.609;
   1:  PR[GP1:91,2] = PR[GP1:90,2] + 93.011;
   1:L PR[91] 10mm/sec FINE;
   1:  PR[GP1:91,1] = PR[GP1:90,1] + 117.840;
   1:  PR[GP1:91,2] = PR[GP1:90,2] + 93.191;
   1:L PR[91] 10mm/sec FINE;
   1:  PR[GP1:91,1] = PR[GP1:90,1] + 119.452;
   1:  PR[GP1:91,2] = PR[GP1:90,2] + 94.669;
   1:L PR[91] 10mm/sec FINE;
   1:  PR[GP1:91,1] = PR[GP1:90,1] + 120.202;
   1:  PR[GP1:91,2] = PR[GP1:90,2] + 95.444;
   1:L PR[91] 10mm/sec FINE;
   1:  PR[GP1:91,1] = PR[GP1:90,1] + 121.019;
   1:  PR[GP1:91,2] = PR[GP1:90,2] + 96.458;
   1:L PR[91] 10mm/sec FINE;
   1:  PR[GP1:91,1] = PR[GP1:90,1] + 122.088;
   1:  PR[GP1:91,2] = PR[GP1:90,2] + 97.934;
   1:L PR[91] 10mm/sec FINE;
   1:  PR[GP1:91,1] = PR[GP1:90,1] + 122.330;
   1:  PR[GP1:91,2] = PR[GP1:90,2] + 98.350;
   1:L PR[91] 10mm/sec FINE;
   1:  PR[GP1:91,1] = PR[GP1:90,1] + 123.058;
   1:  PR[GP1:91,2] = PR[GP1:90,2] + 99.731;
   1:L PR[91] 10mm/sec FINE;
   1:  PR[GP1:91,1] = PR[GP1:90,1] + 123.488;
   1:  PR[GP1:91,2] = PR[GP1:90,2] + 100.491;
   1:L PR[91] 10mm/sec FINE;
   1:  PR[GP1:91,1] = PR[GP1:90,1] + 124.475;
   1:  PR[GP1:91,2] = PR[GP1:90,2] + 103.034;
   1:L PR[91] 10mm/sec FINE;
